			E_PML_Command.Suspend:
				stModeStateOut.RequestedState := E_PML_State.Suspended;
			
			E_PML_Command.Unsuspend:
				stModeStateOut.RequestedState := E_PML_State.Execute;
			
			E_PML_Command.Abort:
				stModeStateOut.RequestedState := E_PML_State.Aborted;
			
			E_PML_Command.Clear:
				stModeStateOut.RequestedState := E_PML_State.Stopped;
			
			E_PML_Command.Complete:
				stModeStateOut.RequestedState := E_PML_State.Complete;
			
		END_CASE

		// Wait done
		IF ((stModeStateOut.RequestedState = eCurrentState) AND (stModeStateOut.ModeStateResponse <= 0)) THEN
			// Set change status
			stModeStateOut.ChangeStatus := stModeStateIn.ChangeRequest;
			stModeStateOut.ModeStateResponse := 3;
			stModeStateOut.DataChange := stModeStateOut.DataChange + 1;
			stModeStateIn.State := E_PML_Command.Undefined;
			eCommand := E_PML_Command.Undefined;
		END_IF
	END_IF
END_IF


// Run State Machine
M_PackML_StateMachine();


// Update current mode/state
IF (DINT_TO_UINT(eCurrentMode) <> stModeStateOut.CurrentMode) THEN
	stModeStateOut.CurrentMode := DINT_TO_UINT(eCurrentMode);
	stModeStateOut.DataChange := stModeStateOut.DataChange + 1;	
END_IF
IF (DINT_TO_UINT(eCurrentState) <> stModeStateOut.CurrentState) THEN
	stModeStateOut.CurrentState := DINT_TO_UINT(eCurrentState);
	stModeStateOut.DataChange := stModeStateOut.DataChange + 1;	
END_IF

/// Static state "Aborted"
/// Trigged by "StateCompleted" when in "Aborting" state
/// Requires "Clear" to go to "Clearing" state 
{attribute 'object_name' := 'M_Aborted'}
METHOD M_Aborted
END_METHOD

/// Dynamic state "Aborting"
/// Trigged by "Abort" command
/// Requires "StateCompleted" to go to "Aborted" state 
{attribute 'object_name' := 'M_Aborting'}
METHOD M_Aborting
M_StateComplete();
END_METHOD

/// Set job data for mechanical roughing
METHOD PROTECTED M_CheckJobData : BOOL
VAR
	i						: UINT;
	bDynamicToolFound		: ARRAY [1..3] OF BOOL;		// Required Dynamic Tool(s) found
	bStationaryToolFound	: ARRAY [1..3] OF BOOL;		// Required Stationary Tool(s) found
	bDynamicMaterialFound	: ARRAY [1..3] OF BOOL;		// Required Dynamic Material(s) found
	bStationaryMaterialFound: ARRAY [1..3] OF BOOL;		// Required Stationary Material(s) found
END_VAR

// Check Job Type
// Should be overwritten in inherited FB's if JobData need to be checked!
M_CheckJobData := TRUE;
END_METHOD

/// Dynamic state "Clearing"
/// Trigged by "Clear" command "Aborted" state
/// Requires "StateCompleted" to go to "Stopped" state 
{attribute 'object_name' := 'M_Clearing'}
METHOD M_Clearing
M_StateComplete();
END_METHOD

/// Static state "Complete"
/// Trigged by "StateCompleted" when in "Completing" state
/// Requires "Reset" to go to "Resetting" state 
{attribute 'object_name' := 'M_Complete'}
METHOD M_Complete
END_METHOD

/// Dynamic state "Completing"
/// Trigged by "StageCompleted" command when in "Execute" state
/// Requires "StateCompleted" to go to "Complete" state 
{attribute 'object_name' := 'M_Completing'}
METHOD M_Completing
M_StateComplete();
END_METHOD

METHOD M_ErrorWarningObj : BOOL
VAR_INPUT
	bActive				: BOOL;
	iErrorWarningType	: UINT;
	diErrorWarningID 	: UDINT;
	sDeviceID			: STRING(30);
	iSeverity			: UINT;
	iNativeID			: UDINT;
	sNativeMessage		: STRING(80);
END_VAR
VAR_IN_OUT
	arErrorWaringData	: ARRAY [1..255] OF ST_ErrorWarningDataX;
END_VAR
VAR
	iFoundPos			: UINT;
	i					: UINT;
	j					: UINT;
END_VAR
//Look through array to find existing record(s)
FOR i := 1 TO 255 DO
	IF arErrorWaringData[i].ErrorWarningID = 0 THEN
		EXIT;
	END_IF
	//Existing alarm - first
	IF arErrorWaringData[i].ErrorWarningID = diErrorWarningID AND iFoundPos = 0 THEN
		iFoundPos := i;
	//Multiple records - delete
	ELSIF arErrorWaringData[i].ErrorWarningID = diErrorWarningID AND iFoundPos <> 0 THEN
		MEMSET(ADR(arErrorWaringData[i]), 0, SIZEOF(arErrorWaringData[i]));
		M_ErrorWarningObj := TRUE;
	END_IF
END_FOR

//Alarm high
IF bActive THEN
	//New alarm
	IF iFoundPos = 0 THEN
		arErrorWaringData[i].ErrorWarningType := iErrorWarningType;
		arErrorWaringData[i].DeviceID := sDeviceID;
		arErrorWaringData[i].Severity := iSeverity;
		arErrorWaringData[i].NativeID := iNativeID;
		arErrorWaringData[i].NativeMessage := sNativeMessage;
		arErrorWaringData[i].ErrorWarningID := diErrorWarningID;
		arErrorWaringData[i].DateTime := SYSTEMTIME_TO_STRING(fbGetTime.TIMESTR);
		M_ErrorWarningObj := TRUE;
	END_IF
	
//Alarm low
ELSIF NOT bActive AND iFoundPos <> 0 THEN
	MEMSET(ADR(arErrorWaringData[iFoundPos]), 0, SIZEOF(arErrorWaringData[iFoundPos]));
	M_ErrorWarningObj := TRUE;
END_IF

//Defrag
IF M_ErrorWarningObj THEN
	FOR i:= 1 TO 254 DO
		//Find first empty spot
		IF arErrorWaringData[i].ErrorWarningID = 0 THEN
			//Find first record
			FOR j:= i TO 255 DO
				IF arErrorWaringData[j].ErrorWarningID <> 0 THEN
					//Move to empty spot
					arErrorWaringData[i] := arErrorWaringData[j];
					MEMSET(ADR(arErrorWaringData[j]), 0, SIZEOF(arErrorWaringData[j]));
					EXIT;
				END_IF
			END_FOR
		END_IF
		//No more records
		IF j >= 255 THEN
			RETURN;
		END_IF
	END_FOR
END_IF
END_METHOD

/// Static state "Execute"
/// Trigged by "StageCompleted" when in "Starting" state
/// Trigged by "StageCompleted" when in "Unholding" state
/// Trigged by "StageCompleted" when in "Unsuspending" state
/// Requires "Hold" command to go to "Holding" state 
/// Requires "Suspend" command to go to "Suspending" state 
/// Requires "StageCompleted" to go to "Completing" state 
{attribute 'object_name' := 'M_Execute'}
METHOD M_Execute
M_StateComplete();
END_METHOD

/// Static state "Held"
/// Trigged by "StateCompleted" when in "Holding" state
/// Requires "Unhold" command to go to "Unholding" state 
{attribute 'object_name' := 'M_Held'}
METHOD M_Held
END_METHOD

/// Dynamic state "Holding"
/// Trigged by "Hold" command when in "Execute" state
/// Requires "StateCompleted" to go to "Held" state 
{attribute 'object_name' := 'M_Holding'}
METHOD M_Holding
M_StateComplete();
END_METHOD

/// Static state "Idle"
/// Trigged by "StateCompleted" when in "Resetting" state
/// Requires "Start" command to go to "Starting" state 
{attribute 'object_name' := 'M_Idle'}
METHOD M_Idle
END_METHOD

METHOD PROTECTED M_Init : BOOL
VAR_INPUT
END_VAR
IF (NOT bInitDone) THEN
	
	// OEE initial values
	stOEE.GoodProduct := iGoodProduct;	
	stOEE.RejectedProduct := iRejectedProduct;	
	stOEE.ProcessedProduct := iProcessedProduct;	

	bInitDone := TRUE;

END_IF
M_Init := bInitDone;
END_METHOD

METHOD PROTECTED M_OEEProductProcessed
VAR_INPUT
	bGood		: BOOL;
END_VAR

// Increment OEE values
iProcessedProduct := iProcessedProduct + 1;
stOEE.ProcessedProduct := iProcessedProduct;
IF (bGood) THEN
	iGoodProduct := iGoodProduct + 1;
	stOEE.GoodProduct := iGoodProduct;
ELSE
	iRejectedProduct := iRejectedProduct + 1;
	stOEE.RejectedProduct := iRejectedProduct;
END_IF

// TODO!!!
// Update Event ID!
stOEE.EventID;

// Update time for changes
stOEE.DateTime := SYSTEMTIME_TO_DT(TIMESTR := fbGetTime.TIMESTR);

// Increment DataChange to signal to LC that sometihng has changed
stOEE.DataChange := stOEE.DataChange + 1;
END_METHOD

METHOD PROTECTED M_PackML_StateMachine : BOOL
VAR_INPUT
END_VAR

CASE nStateModeChange OF

	0:	// Waiting for user request
		IF (NOT UnitModeChangeInProcess) THEN
			// Local unit mode change request
			IF (bProductionLocal AND (eCurrentMode <> Tc3_PackML_V2.ePMLProtUnitMode_Production)) THEN
				eMode := E_PML_Mode.Production;
				UnitModeChangeRequest := TRUE;
			ELSIF (bManualLocal AND (eCurrentMode <> Tc3_PackML_V2.ePMLProtUnitMode_Manual)) THEN
				eMode := E_PML_Mode.Manual;
				UnitModeChangeRequest := TRUE;
			ELSIF (bMaintenanceLocal AND (eCurrentMode <> Tc3_PackML_V2.ePMLProtUnitMode_Maintenance)) THEN
				eMode := E_PML_Mode.Maintenance;
				UnitModeChangeRequest := TRUE;
			END_IF
		END_IF
		bChangeIntoProduction := FALSE;
		IF ((eMode = ePMLProtUnitMode_Production) AND (eCurrentMode = ePMLProtUnitMode_Invalid)) THEN
			nStateModeChange := 1;
		ELSIF (UnitModeChangeRequest AND (eMode <> ePMLProtUnitMode_Production)) THEN
			nStateModeChange := 1;
		ELSIF ((eMode = ePMLProtUnitMode_Production) AND (eCurrentMode <> ePMLProtUnitMode_Production)) THEN
			nStateModeChange := 3;
		END_IF
		
	1:	// Starting UnitModeManager 
		fbUnitModeManager.bExecute := TRUE;
		fbUnitModeManager.eModeCommand := eMode;
		UnitModeChangeInProcess := TRUE;
	
		IF (fbUnitModeManager.bDone) THEN
			fbUnitModeManager.bExecute := FALSE;
			bInvalidModeCommandOut := FALSE;
			nStateModeChange := 0;
			bChangeIntoProduction := FALSE;
			UnitModeChangeInProcess := FALSE;
		ELSIF (fbUnitModeManager.bError) THEN
			bInvalidModeCommandOut := TRUE;
			fbUnitModeManager.bExecute := FALSE;
			nLastState := eCurrentState;
			nStateModeChange := 2;
			bChangeIntoProduction := FALSE;
			UnitModeChangeInProcess := FALSE;
		END_IF
	
	2:	// ErrorHanddling
		IF (bModeChangeRequest) THEN
			nStateModeChange := 0;
			bInvalidModeCommandOut := FALSE;
		ELSIF (nLastState <> eCurrentState) THEN
			bInvalidModeCommandOut := FALSE;
		END_IF
		
	3:	// state to check, if command 'Production' is valid
		IF ((eCurrentState = ePMLState_Aborted) OR (eCurrentState = ePMLState_Stopped) OR (eCurrentState = ePMLState_Idle)) THEN
			bChangeIntoProduction := TRUE;
			nStateModeChange := 1;
		ELSE
			nStateModeChange := 2;
			bInvalidModeCommandOut := TRUE;
			nLastState := eCurrentState;
		END_IF
END_CASE


// Run Unit Mode Manager
fbUnitModeManager(	eState := eCurrentState,
					eModeStatus => eCurrentMode,
					bDone => ,
					bError => ,
					nErrorId => 	);

IF (fbUnitModeManager.eModeStatus <> 0) THEN
	// Local E-stop/abort handling	
	IF (NOT bEStopOK OR bAbortLocal) THEN
		eCommand := DINT_TO_UINT(E_PMLCommand.ePMLCommand_Abort);
	END_IF
	// Local Start handling
	IF (bStartLocal) THEN
		eCommand := DINT_TO_UINT(E_PMLCommand.ePMLCommand_Start);
	END_IF
	// Local Stop handling
	IF (bStopLocal) THEN
		eCommand := DINT_TO_UINT(E_PMLCommand.ePMLCommand_Stop);
	END_IF
	// Local Reset handling
	IF (bResetLocal) THEN
		eCommand := DINT_TO_UINT(E_PMLCommand.ePMLCommand_Reset);
	END_IF
	// Local Clear handling
	IF (bClearLocal) THEN
		eCommand := DINT_TO_UINT(E_PMLCommand.ePMLCommand_Clear);
	END_IF
	// Local Hold handling
	IF (bHoldLocal) THEN
		eCommand := DINT_TO_UINT(E_PMLCommand.ePMLCommand_Hold);
	END_IF
	// Local Unhold handling
	IF (bUnholdLocal) THEN
		eCommand := DINT_TO_UINT(E_PMLCommand.ePMLCommand_Unhold);
	END_IF
	// Local Suspend handling
	IF (bSuspendLocal) THEN
		eCommand := E_PMLCommand.ePMLCommand_Suspend;
	END_IF
	// Local Unsuspend handling
	IF (bSuspendLocal) THEN
		eCommand := E_PMLCommand.ePMLCommand_Unsuspend;
	END_IF
	
	// Calling the StateMachine, when there is a valid Mode
	fbStateMachine(	eMode := eCurrentMode,
					eCommand := eCommand,
					stSubUnitInfoRef := ,
					stOptions := ,
					eState => eCurrentState,
					bError => ,
					nErrorID => 	);

END_IF

// Requested state:
CASE eCommand OF			
	E_PMLCommand.ePMLCommand_Abort:
		eRequestedState := E_PMLState.ePMLState_Aborted;
		
	E_PMLCommand.ePMLCommand_Clear:
		eRequestedState := E_PMLState.ePMLState_Stopped;

	E_PMLCommand.ePMLCommand_Complete:
		eRequestedState := E_PMLState.ePMLState_Complete;
		
	E_PMLCommand.ePMLCommand_Hold:
		eRequestedState := E_PMLState.ePMLState_Held;
		
	E_PMLCommand.ePMLCommand_Reset:
		eRequestedState := E_PMLState.ePMLState_Idle;
		
	E_PMLCommand.ePMLCommand_Start:
		eRequestedState := E_PMLState.ePMLState_Execute;
		
	E_PMLCommand.ePMLCommand_Stop:
		eRequestedState := E_PMLState.ePMLState_Stopped;
		
	E_PMLCommand.ePMLCommand_Suspend:
		eRequestedState := E_PMLState.ePMLState_Suspended;
		
	E_PMLCommand.ePMLCommand_Unhold:
		eRequestedState := E_PMLState.ePMLState_Execute;
		
	E_PMLCommand.ePMLCommand_Unsuspend:
		eRequestedState := E_PMLState.ePMLState_Execute;
		
END_CASE


//One of the methods is executing by the actual state
CASE eCurrentState OF
	E_PML_State.Undefined:
		M_Undefined();
	E_PML_State.Clearing:
		M_Clearing();
	E_PML_State.Stopped:
		M_Stopped();
	E_PML_State.Starting:
		M_Starting();
	E_PML_State.Idle:
		M_Idle();
	E_PML_State.Suspended:
		M_Suspended();
	E_PML_State.Execute:
		M_Execute();
	E_PML_State.Stopping:
		M_Stopping();
	E_PML_State.Aborting:
		M_Aborting();
	E_PML_State.Aborted:
		M_Aborted();
	E_PML_State.Holding:
		M_Holding();
	E_PML_State.Held:
		M_Held();
	E_PML_State.Unholding:
		M_Unholding();
	E_PML_State.Suspending:
		M_Suspending();
	E_PML_State.Unsuspending:
		M_Unsuspending();
	E_PML_State.Resetting:
		M_Resetting();
	E_PML_State.Completing:
		M_Completing();
	E_PML_State.Complete:
		M_Complete();
END_CASE
END_METHOD

/// Dynamic state "Resetting"
/// Trigged by "Reset" command when in "Stopped" state
/// Requires "StateCompleted" to go to "Idle" state 
{attribute 'object_name' := 'M_Resetting'}
METHOD M_Resetting
M_StateComplete();
END_METHOD

/// Dynamic state "Starting"
/// Trigged by "Start" command when in "Idle" state
/// Requires "StateCompleted" to go to "Execute" state 
{attribute 'object_name' := 'M_Starting'}
METHOD M_Starting
M_StateComplete();
END_METHOD

{attribute 'object_name' := 'M_StateComplete'}
METHOD M_StateComplete
//the actual state is completed
fbStateMachine.M_StateComplete();
END_METHOD

/// Static state "Stopped"
/// Trigged by "StateCompleted" when in "Stopping" state
/// Requires "Reset" command to go to "Resetting" state 
{attribute 'object_name' := 'M_Stopped'}
METHOD M_Stopped
END_METHOD

/// Dynamic state "Stopping"
/// Trigged by "Stop" command
/// Requires "StateCompleted" to go to "Stopped" state 
{attribute 'object_name' := 'M_Stopping'}
METHOD M_Stopping
M_StateComplete();
END_METHOD

/// Static state "Suspended"
/// Trigged by "StateCompleted" when in "Suspending" state
/// Requires "Unsuspend" command to go to "Unsuspending" state 
{attribute 'object_name' := 'M_Suspended'}
METHOD M_Suspended
END_METHOD

/// Dynamic state "Suspending"
/// Trigged by "Suspend" command when in "Execute" state
/// Requires "StateCompleted" to go to "Suspended" state 
{attribute 'object_name' := 'M_Suspending'}
METHOD M_Suspending
M_StateComplete();
END_METHOD

{attribute 'object_name' := 'M_Undefined'}
METHOD M_Undefined
END_METHOD

/// Dynamic state "Unholding"
/// Trigged by "Unhold" command when in "Held" state
/// Requires "StateCompleted" to go to "Execute" state 
{attribute 'object_name' := 'M_Unholding'}
METHOD M_Unholding
M_StateComplete();
END_METHOD

/// Dynamic state "Unsuspending"
/// Trigged by "Unsuspend" command when in "Suspended" state
/// Requires "StateCompleted" to go to "Execute" state 
{attribute 'object_name' := 'M_Unsuspending'}
METHOD M_Unsuspending
M_StateComplete();
END_METHOD

END_FUNCTION_BLOCK

// ---- ECC/Tools/F_LogLine.TcPOU
FUNCTION F_LogLine : DINT
VAR_INPUT
	sLogString	: STRING(250);
	iValue		: DINT;
END_VAR
VAR
	iReplacePos	: INT;
	sLogFile	: STRING;
END_VAR

	// Log to output window as info message
	IF (bLogToOutputWindow) THEN
		F_LogLine:= ADSLOGDINT(ADSLOG_MSGTYPE_HINT OR ADSLOG_MSGTYPE_LOG,sLogString, iValue);
	END_IF
	
	// Replace the '%d' in the log string with the stinr-value of the iValue input 
	iReplacePos := FIND(sLogString, '%d');
	IF (iReplacePos > 0) THEN
		// '%d' found in string
		sLogFile := REPLACE(sLogString, DINT_TO_STRING(iValue), 2, iReplacePos);
	ELSE
		sLogFile := sLogString;
	END_IF

	// Log to file
	F_LogFile(sLogFile);

END_FUNCTION

// ---- ECC/Tools/LogToFile/F_LogFile.TcPOU
FUNCTION F_LogFile : BOOL
VAR_INPUT
	msg		: STRING(200);

END_VAR
VAR
	Temp:ULINT;
	CurrentDate:STRING(10);
	msgWithTime :STRING(200);
	DateTimeNow :STRING;
END_VAR

(* Get date and time *)

DateTimeNow  := SYSTEMTIME_TO_STRING(fbLocalTime.systemTime);

(* Set date to check for generation of new file *)
CurrentDate := DateTimeNow;

(* Add date and time to line of log *)
msgWithTime := CONCAT(DateTimeNow, ' ');
msgWithTime := CONCAT(msgWithTime, msg);
msgWithTime := CONCAT(msgWithTime, '$N');


(* Write to FIFO *)
IF LogToTextBuffer.Count <= LogToTextBuffer.DataTop THEN

	(* Calculate new insert pointer *)
	LogToTextBuffer.Input_Pointer := LogToTextBuffer.Input_Pointer + 1;
	IF LogToTextBuffer.Input_Pointer > LogToTextBuffer.DataTop THEN
		LogToTextBuffer.Input_Pointer := 0;
	END_IF

	(* If data is empty, sync output pointer *)
	IF LogToTextBuffer.Count = 0 THEN
		LogToTextBuffer.Output_Pointer := LogToTextBuffer.Input_Pointer;
	END_IF

	(* Store data *)
	LogToTextBuffer.DB[LogToTextBuffer.Input_Pointer] := msgWithTime;

	LogToTextBuffer.Count := LogToTextBuffer.Count + 1;
END_IF

END_FUNCTION

// ---- ECC/Cell_Unit_4/HeatAndSteamDeviceDriver/FB_EMS_HS.TcPOU
FUNCTION_BLOCK FB_EMS_HS
VAR_INPUT
END_VAR
VAR_OUTPUT
END_VAR
VAR
// ModBus data structures
	uRead			: U_EMS_HS_Read;
	uWrite			: U_EMS_HS_Write;
	
	// Modbus reading
	tonMBRead		: TON;		// Timer to handle reading requests from device
	fbMBRead		: Tc2_ModbusSrv.FB_MBReadRegs;	// FB for reading modbus register(s)
	bMBRead_Busy	: BOOL;
	bMBRead_Error	: BOOL;
	nMBRead_ErrorID	: UDINT;
	cbMBRead_Read	: UDINT;
	trigMBReadError	: R_TRIG;
	fbGetReadTime	: NT_GetTime;
	trigReadDone	: F_TRIG;
	tsLastRead		: TIMESTRUCT;
	iReads			: UINT;
	iErrorReads		: UINT;

// Modbus writing
	tonMBWrite		: TON;		// Timer to handle writing requests to device
	fbMBWrite		: Tc2_ModbusSrv.FB_MBWriteRegs;	// FB for writing modbus register(s)
	bMBWrite_Busy	: BOOL;
	bMBWrite_Error	: BOOL;
	nMBWrite_ErrorID: UDINT;
	trigWriteDone	: F_TRIG;
	trigMBWriteError: R_TRIG;
	fbGetWriteTime	: NT_GetTime;
	tsLastWrite		: TIMESTRUCT;
	iWrites			: UINT;
	iErrorWrites	: UINT;
	
//Local vars
	bAbortLocal 	: BOOL;
	bManualLocal	: BOOL;
	bProductionLocal: BOOL;
// Simulation
	bSimMode		: BOOL;	// TRUE if simulation should be used (no start device, no setpoints to device)
END_VAR
VAR PERSISTENT
	sIPAddr			: STRING(15);	// Station IP address
	tTimeout		: TIME := T#5S;
END_VAR


// Simulation mode ?
// Only perform communication if NOT in simulation mode
IF (NOT M_Simulation()) THEN

	// Device controller
	M_ModBusRead(	rInterval := 1,
					wAddress := 2501,
					wNoOfRegisters := 23,
					pbDestAddress := ADR(uRead.aWords),
					dwDestSize := SIZEOF(uRead.aWords)	);
	
	M_ModBusWrite(	rInterval := 1, 
					wAddress := 2601,
					wNoOfRegisters := 8,	
					pbSrcAddress := ADR(uWrite.aWords),
					dwSrcSize := SIZEOF(uWrite.aWords)	);
END_IF

// Local state changes
IF (uRead.stVars.eMachStatus = E_EMS_HS_Status.ALARM) THEN
	bAbortLocal := TRUE;
ELSIF (uRead.stVars.stStates.ALARM_IN_PROGRESS) THEN
	bAbortLocal := TRUE;
ELSIF (NOT uRead.stVars.stStates.REMOTE_MODE) THEN
	bAbortLocal := TRUE;
ELSE
	bAbortLocal := FALSE;
END_IF
IF (NOT uRead.stVars.stStates.REMOTE_MODE) THEN
	bManualLocal := TRUE;
	bProductionLocal := FALSE;
ELSE
	bProductionLocal := TRUE;
	bManualLocal := FALSE;
END_IF

METHOD PROTECTED M_CmdNeutral : BOOL
VAR_INPUT
END_VAR
uWrite.stVars.stCommands.REMOTE_START := FALSE;
uWrite.stVars.stCommands.REMOTE_STOP := FALSE;
END_METHOD

METHOD PROTECTED M_Cmdreset : BOOL
VAR_INPUT
END_VAR
END_METHOD

METHOD PROTECTED M_CmdStart : BOOL
VAR_INPUT
END_VAR
uWrite.stVars.stCommands.REMOTE_START := TRUE;
uWrite.stVars.stCommands.REMOTE_STOP := FALSE;
END_METHOD

METHOD PROTECTED M_CmdStop : BOOL
VAR_INPUT
END_VAR
uWrite.stVars.stCommands.REMOTE_START := FALSE;
uWrite.stVars.stCommands.REMOTE_STOP := TRUE;
END_METHOD

/// Read modbus TCP register(s)
METHOD PROTECTED M_ModBusRead : BOOL
VAR_INPUT
	rInterval		: REAL;
	wAddress		: WORD;				// Register address to read
	wNoOfRegisters	: WORD;				// Register to read from station
	pbDestAddress	: POINTER TO BYTE;	// Address of mem to place read data
	dwDestSize		: DWORD;			// Size of mem to place read data
END_VAR
// Timer
tonMBRead(	IN := NOT tonMBRead.Q,
			PT := REAL_TO_TIME(rInterval * 1000.0),
			Q => 	);

// Read data from device via. modbus TCP
fbMBRead(	sIPAddr:= sIPAddr, 				// Station IP address
			nTCPPort:= MODBUS_TCP_PORT, 	// Modbus TCP port (normally 502)
			nUnitID:= 1,//16#FF, 			// If a device is addressed directly via TCP/IP, this value must be 16#FF.
			nQuantity:= wNoOfRegisters,		// Number of words (registers) to read 
			nMBAddr:= wAddress - 1,			// Addres of registers to read ( -1 needed ) 
			cbLength:= dwDestSize,			// Contains the max. byte size of the destination buffer. The minimum buffer byte size must be: nQuantity * 2.
			pDestAddr:= pbDestAddress, 		// Address of the destination buffer into which the data are to be read.
			bExecute:= tonMBRead.Q,			// Trig reading
			tTimeout:= tTimeout, 			// States the length of the timeout that may not be exceeded by execution of the ADS command
			bBusy=> bMBRead_Busy, 
			bError=> bMBRead_Error, 
			nErrId=> , 
			cbRead=> cbMBRead_Read);

// Last read time
trigReadDone(CLK := (fbMBRead.bBusy AND NOT fbMBRead.bError));
trigMBReadError(CLK := bMBRead_Error);
IF (trigReadDone.Q) THEN
	iReads := iReads + 1;
END_IF
IF (trigMBReadError.Q) THEN
	iErrorReads := iErrorReads + 1;
	nMBRead_ErrorID := fbMBRead.nErrId;
END_IF
fbGetReadTime(	NETID:= '', 
				START:= trigReadDone.Q,
				TMOUT:= T#5S, 
				BUSY=> , 
				ERR=> , 
				ERRID=> , 
				TIMESTR=> tsLastRead);

// Station communication status
M_ModBusRead := (cbMBRead_Read = wNoOfRegisters * 2);
END_METHOD

/// Writes ModBus TCP registers
METHOD PROTECTED M_ModBusWrite : BOOL
VAR_INPUT
	rInterval		: REAL;
	wAddress		: WORD;				// Register address to write to
	wNoOfRegisters	: WORD;				// Register(s) to write to station
	pbSrcAddress	: POINTER TO BYTE;	// Address of mem to read source data from
	dwSrcSize		: DWORD;			// Size of mem to read source data from
END_VAR
VAR
END_VAR
// Timer
tonMBWrite(	IN := NOT tonMBWrite.Q,
			PT := REAL_TO_TIME(rInterval * 1000.0),
			Q => 	);

// Write data to device via. modbus TCP
fbMBWrite(	sIPAddr:= sIPAddr, 				// Station IP address
			nTCPPort:= MODBUS_TCP_PORT, 	// Modbus TCP port (normally 502)
			nUnitID:= 1,//16#FF, 			// If a device is addressed directly via TCP/IP, this value must be 16#FF.
			nQuantity:= wNoOfRegisters,		// Number of words (registers) to write 
			nMBAddr:= wAddress - 1,			// Addres of registers to write 
			cbLength:= dwSrcSize,			// Contains the max. byte size of the source buffer. The minimum buffer byte size must be: nQuantity * 2.
			pSrcAddr:= pbSrcAddress,	 	// Address of the source buffer from which, the data are read
			bExecute:= tonMBWrite.Q,		// Trig writing 
			tTimeout:= tTimeout, 			// States the length of the timeout that may not be exceeded by execution of the ADS command
			bBusy=> bMBWrite_Busy, 
			bError=> bMBWrite_Error, 
			nErrId=> );

// Last write time
trigWriteDone(CLK := (fbMBWrite.bBusy AND NOT fbMBWrite.bError));
trigMBWriteError(CLK := bMBWrite_Error);
IF (trigWriteDone.Q) THEN
	iWrites := iWrites + 1;
END_IF
IF (trigMBWriteError.Q) THEN
	iErrorWrites := iErrorWrites + 1;
	nMBWrite_ErrorID := fbMBWrite.nErrId;
END_IF
fbGetWriteTime(	NETID:= '', 
				START:= trigWriteDone.Q,
				TMOUT:= T#5S, 
				BUSY=> , 
				ERR=> , 
				ERRID=> , 
				TIMESTR=> tsLastWrite);

// Station communication status
M_ModBusWrite := trigWriteDone.Q;
END_METHOD

METHOD PROTECTED M_Simulation : BOOL
VAR_INPUT
END_VAR

IF (bSimMode) THEN
	// Simulation mode ENABLED

	// Device start command
	IF (uWrite.stVars.stCommands.REMOTE_START) THEN
		// Device states
		uRead.stVars.eMachStatus := E_EMS_HS_Status.READY;
		uRead.stVars.stStates.MACHINE_READY_TO_WORK := TRUE;
		uRead.stVars.stStates.TEMP_START_BELT_REACHED := TRUE;
		uRead.stVars.stStates.TEMP_START_STEAM_REACHED := TRUE;
		uRead.stVars.stStates.MACHINE_IN_STANDBY := FALSE;
		// Device temperature
		uRead.stVars.rActTempVal := uWrite.stVars.rSetTemp;
	ELSE
		// Device states
		uRead.stVars.eMachStatus := E_EMS_HS_Status.STANDBY;
		uRead.stVars.stStates.MACHINE_READY_TO_WORK := FALSE;
		uRead.stVars.stStates.TEMP_START_BELT_REACHED := FALSE;
		uRead.stVars.stStates.TEMP_START_STEAM_REACHED := FALSE;
		uRead.stVars.stStates.MACHINE_IN_STANDBY := TRUE;
	END_IF
	// Temperature setpoint value
	uRead.stVars.rActTempSetpoint := uWrite.stVars.rSetTemp;
	// Steam setpoint value
	uRead.stVars.rActSteamReq := uWrite.stVars.rSetSteamReq;
	// Fan setpoint value
	uRead.stVars.rActFanReq := uWrite.stVars.rSetFanSpeed;
	// Alarms
	uRead.stVars.stAlarms.TEMP_PROBE_FAULT := FALSE;
	uRead.stVars.stAlarms.FAULT_INVERTER := FALSE;
	uRead.stVars.stAlarms.ENERGY_METER_COM_ERROR := FALSE;
	// Device states
	uRead.stVars.stStates.REMOTE_MODE := TRUE;
	uRead.stVars.stStates.ALARM_IN_PROGRESS := FALSE;
	uRead.stVars.stStates.MACHINE_IN_HEATING := FALSE;
	
	M_Simulation := TRUE;

ELSE
	// Simulation mode DISABLED

	M_Simulation := FALSE;

END_IF
END_METHOD

METHOD PROTECTED M_StaAlarm : BOOL
VAR_INPUT
END_VAR
M_StaAlarm := (uRead.stVars.eMachStatus = E_EMS_HS_Status.ALARM);
END_METHOD

METHOD PROTECTED M_StaReady : BOOL
VAR_INPUT
END_VAR
M_StaReady := (uRead.stVars.eMachStatus = E_EMS_HS_Status.READY);
END_METHOD

METHOD PROTECTED M_StaStandby : BOOL
VAR_INPUT
END_VAR
M_StaStandby := (uRead.stVars.eMachStatus = E_EMS_HS_Status.STANDBY);
END_METHOD

PROPERTY PUBLIC P_bSimulationMode : BOOL
GET
P_bSimulationMode := bSimMode;
END_GET
SET
bSimMode := P_bSimulationMode;
END_SET
END_PROPERTY

PROPERTY P_ModbusIPBarrera : STRING
GET
P_ModbusIPBarrera := sIPAddr;
END_GET
SET
sIPAddr := P_ModbusIPBarrera;
END_SET
END_PROPERTY

PROPERTY PUBLIC P_rSetFanSpeed : REAL
SET
uWrite.stVars.rSetFanSpeed := P_rSetFanSpeed;
END_SET
END_PROPERTY

PROPERTY PUBLIC P_rSetSteamReq : REAL
SET
uWrite.stVars.rSetSteamReq := REAL_TO_DINT(P_rSetSteamReq);
END_SET
END_PROPERTY

PROPERTY PUBLIC P_rSetTemp : REAL
SET
uWrite.stVars.rSetTemp := P_rSetTemp;
END_SET
END_PROPERTY

PROPERTY PUBLIC P_stCellCommandData : ST_EMS_HS_Write
GET // PUBLIC
P_stCellCommandData := uWrite.stVars;
END_GET
SET // PUBLIC
uWrite.stVars := P_stCellCommandData;
END_SET
END_PROPERTY

PROPERTY PUBLIC P_stCellStatusData : ST_EMS_HS_Read
GET
P_stCellStatusData := uRead.stVars;
END_GET
END_PROPERTY

END_FUNCTION_BLOCK

// ---- ECC/Tools/F_StringCompNoCase.TcPOU
FUNCTION F_StringCompNoCase : BOOL
VAR_INPUT
	s1		: STRING;
	s2		: STRING;
END_VAR
VAR
END_VAR


F_StringCompNoCase := ( F_ToUCase(s1) = F_ToUCase(s2) );

END_FUNCTION

// ---- ECC/Basic/OPC Data/F_NewDeviceDataX.TcPOU
FUNCTION F_NewDeviceDataX : ST_DeviceDataX
VAR_INPUT
	sDeviceID			: STRING;			// The ID of the specific device
	sDeviceName			: STRING;			// The descriptive name of the device
	iDataID				: UDINT;			// The ID of the operational data
	sDataName			: STRING;			// The descriptive name of the operational data
	eUnit				: E_Units;	// The symbolic description of the measuring unit
END_VAR
VAR
END_VAR

// Create structure

F_NewDeviceDataX.DeviceID := sDeviceID;
F_NewDeviceDataX.DeviceName :=sDeviceName;
F_NewDeviceDataX.DataID := iDataID;
F_NewDeviceDataX.DataName := sDataName;
F_NewDeviceDataX.UnitID := Units.Code(eUnit);	// Extracts common unit code from pre-defined unit types
F_NewDeviceDataX.Unit := Units.Text(eUnit);		// Extracts common unit symbol from pre-definded unit types

END_FUNCTION

// ---- ECC/Cell_Unit_4/HeatAndSteam/F_CalcValuesHeatSteam.TcPOU
FUNCTION F_CalcValuesHeatSteam : REAL
VAR_INPUT
	rTempFinal		: REAL;				// [°C]		
	rTempInitial	: REAL;				// [°C]		
	rCT				: REAL;				// []		Coefficient for temperature
	rCS				: REAL;				// []		Coefficient for steam
	rCA				: REAL;				// []		Coefficient for airflow
	rMachineLength	: REAL;				// [m]		Length of machine
	// Limits
	rTimeMin		: REAL;				// [s]		Minimum allowed time in machine
	rTimeMax		: REAL;				// [s]		Maximum allowed time in machine
	rTempMin		: REAL;				// [°C]		Minimum allowed temperature in machine
	rTempMax		: REAL;				// [°C]		Maximum allowed temperature in machine
	rSteamMin		: REAL;				// []		Minimum allowed steam in machine
	rSteamMax		: REAL;				// []		Maximum allowed steam in machine
	rAirMin			: REAL;				// []		Minimum allowed airflow in machine
	rAirMax			: REAL;				// []		Maximum allowed airflow in machine	
END_VAR
VAR_OUTPUT
	rVelocity		: REAL;				// [m/s]	Carrier velocity
	rTempMachine	: REAL;				// [°C]		Machine temperature
	rTimeMachine	: REAL;				// [s]		Time in machine
	rSteamMachine	: REAL;				// []		
	rAirMachine		: REAL;				// []		
END_VAR
VAR
	// Limits
	rVelocityMin	: REAL := 0.001;	// [m/s]	Minimum allowed speed
	rVelocityMax	: REAL := 2.0;		// [m/s]	Maximum allowed speed
	
	// Temp
	rVelocityCalcRaw: REAL;				// [m/s]	
	rVelocityCalc	: REAL;				// [m/s]	
	rTimeCalcRaw	: REAL;				// [s]		
	rTimeCalc		: REAL;				// [s]		
	sTempString		: STRING(200);		// 			
END_VAR


// Calculate time needed in device and machine temperature
//t = ( (TFinal) / (TMachine * cT + SMachine * cS + AMachine * cA) ) - TInitial

// If constants are ZERO use fixed time in mechine from job data (minimum time)
IF ( (rCT = 0.0) AND (rCS = 0.0) AND (rCA = 0.0) ) THEN
	rTimeCalcRaw := rTimeMin;
	rTempMachine := rTempMax;
	rSteamMachine := rSteamMax;
	rAirMax := rAirMax;
	
ELSE
	rTempMachine := (rTempMin + rTempMax) / 2.0;
	rSteamMachine := (rSteamMin + rSteamMax) / 2.0;
	rAirMachine := (rAirMin + rAirMax) / 2.0;

	// Check for divide-by-zero
	IF ((rTempMachine * rCT) + (rSteamMachine * rCS) + (rAirMachine * rCA)) = 0.0 THEN
		rTimeCalcRaw := rTimeMin;
		rTempMachine := rTempMax;
		rSteamMachine := rSteamMax;
		rAirMax := rAirMax;
	ELSE
		rTimeCalcRaw := (rTempFinal - rTempInitial) / ((rTempMachine * rCT) + (rSteamMachine * rCS) + (rAirMachine * rCA));	
	END_IF
	
END_IF

// Limit time in device according to job data
rTimeCalc := LIMIT(rTimeMin, rTimeCalcRaw, rTimeMax);

// Make sure time is not ZERO
IF (rTimeCalc <= 0.0) THEN
	rTimeCalc := 120.0;

END_IF

// Calculate velocity based on time in machine and machine length
rVelocityCalcRaw := rMachineLength / rTimeCalc;

// Limit velocity to allowed limits
rVelocityCalc := LIMIT(rVelocityMin, rVelocityCalcRaw, rVelocityMax);

// Log
	sTempString := CONCAT('STAT: ', 'Velocity Calc ');
	sTempString := CONCAT(sTempString, '. Temp=');
	sTempString := CONCAT(sTempString, TO_STRING(rTempMachine));
	sTempString := CONCAT(sTempString, '. Steam=');
	sTempString := CONCAT(sTempString, TO_STRING(rSteamMachine));
	sTempString := CONCAT(sTempString, '. Air=');
	sTempString := CONCAT(sTempString, TO_STRING(rAirMachine));
	sTempString := CONCAT(sTempString, '. Time_RAW=');
	sTempString := CONCAT(sTempString, TO_STRING(rTimeCalcRaw));
	sTempString := CONCAT(sTempString, '. Time=');
	sTempString := CONCAT(sTempString, TO_STRING(rTimeCalc));
	sTempString := CONCAT(sTempString, '. Vel_RAW=');
	sTempString := CONCAT(sTempString, TO_STRING(rVelocityCalcRaw));
	sTempString := CONCAT(sTempString, '. Vel=');
	sTempString := CONCAT(sTempString, TO_STRING(rVelocityCalc));
	F_Logfile(sTempString);

// Output
rVelocity := rVelocityCalc;
rTempMachine := rTempMachine;
rSteamMachine := rSteamMachine;
rAirMachine := rAirMachine;
rTimeMachine := rTimeCalc;

END_FUNCTION

// ---- ECC/Cell_Unit_4/HeatAndSteam/FB_HeatAndSteamOUT.TcPOU
FUNCTION_BLOCK FB_HeatAndSteamOUT EXTENDS FB_Station_Basic
VAR_INPUT
END_VAR
VAR_OUTPUT
END_VAR
VAR_IN_OUT
	// Inputs
	stJobDataIn				: ST_InputStationHSJobData;
	stConfigIn				: ST_InputStationHSConfiguration;
	stUpcomingConfigIn		: ST_InputStationHSUpcomingConfiguration;
	stControlIn				: ST_InputStationHSControl;
	stAdditionalDataIn		: ST_InputStationHSAdditionalData;
	// Outputs
	stJobDataOut			: ST_OutputStationHSJobData;
	stConfigOut				: ST_OutputStationHSCurrentConfiguration;
	stUpcomingConfigOut		: ST_OutputStationHSUpcomingConfiguration;
	stOperationalDataOut	: ST_OutputStationHSOperationalData;
	stSustainabilityData	: ST_OutputStationHSSustainabilityData;
	stAdditionalDataOut		: ST_OutputStationHSAdditionalData;	
END_VAR 
VAR
	iOldChangeRequest		: UINT;

// Start up
	nCheckValid				: UINT;

END_VAR

SUPER^( stModeStateIn := stModeStateIn,
		stModeStateOut := stModeStateOut,
		stOEE := stOEE,
		stErrorWarning := stErrorWarning);

M_Init();

//Automatic reset when operation complete
bResetLocal := (eCommand <> ePMLCommand_Start AND eCurrentState = E_PMLState.ePMLState_Complete);

/// Static state "Aborted"
/// Trigged by "StateCompleted" when in "Aborting" state
/// Requires "Clear" to go to "Clearing" state 
{attribute 'object_name' := 'M_Aborted'}
METHOD M_Aborted
END_METHOD

/// Dynamic state "Aborting"
/// Trigged by "Abort" command
/// Requires "StateCompleted" to go to "Aborted" state 
{attribute 'object_name' := 'M_Aborting'}
METHOD M_Aborting
// Stop all moving parts
(* STOP all OPSTIONS and Track - Clear alarms og gå til Complete*)

M_StateComplete();
END_METHOD

METHOD M_ClearAll : BOOL
VAR_INPUT
END_VAR

IF eCurrentState = E_PMLState.ePMLState_Aborted OR eCurrentState = E_PMLState.ePMLState_Aborting THEN
	
	F_Logfile('ST2 - All data cleared!');
	
	M_ClearAll := TRUE;
END_IF
END_METHOD

/// Dynamic state "Clearing"
/// Trigged by "Clear" command "Aborted" state
/// Requires "StateCompleted" to go to "Stopped" state 
{attribute 'object_name' := 'M_Clearing'}
METHOD M_Clearing
(* Clear all OPSTIONS and Track - Clear alarms og gå til Complete*)

M_StateComplete();
END_METHOD

/// Static state "Complete"
/// Trigged by "StateCompleted" when in "Completing" state
/// Requires "Reset" to go to "Resetting" state 
{attribute 'object_name' := 'M_Complete'}
METHOD M_Complete
END_METHOD

/// Dynamic state "Completing"
/// Trigged by "StageCompleted" command when in "Execute" state
/// Requires "StateCompleted" to go to "Complete" state 
{attribute 'object_name' := 'M_Completing'}
METHOD M_Completing

VAR
	
END_VAR

// Reset execute sequence
// Job status data to OPC 

//Store old data for comparison



M_StateComplete();
END_METHOD

METHOD M_ConfigurationHandling
VAR_INPUT
END_VAR
VAR
	sTempSTring		: STRING(200);
END_VAR
// Is updated from operator/HMI
IF (stConfigIn.ChangeRequest <> stConfigOut.ChangeStatus) AND (stConfigIn.ChangeRequest > 0) THEN
	sTempString := CONCAT('Station 2 - ConfigChange request - Old request: ', TO_STRING(stConfigOut.ChangeStatus));
	sTempString := CONCAT(sTempString, ', New request: ');
	sTempString := CONCAT(sTempString, TO_STRING(stConfigIn.ChangeRequest));
	sTempString := CONCAT(sTempString, ' ConfigType: ');
	F_LogFile(CONCAT(sTempString, stConfigIn.ConfigurationType)); 
	
	// Change request from Line Controller
	stConfigOut.ChangeAcknowledge := stConfigIn.ChangeRequest;
	
	// Check Configuration Type
	IF (stConfigIn.ConfigurationType = 'OP11600') THEN	
		// Update output job data
		stConfigOut.ConfigurationType := stConfigIn.ConfigurationType;
		stConfigOut.DateTime := SYSTEMTIME_TO_DT(timestr:=fbGetTime.TIMESTR);
		stConfigOut.OP11600 := stConfigIn.OP11600;
		
		// Signal that job data has been written		
		stConfigOut.ChangeStatus := stConfigIn.ChangeRequest;
		
		// Signal that output job data has been updated
		stConfigOut.DataChange := stConfigOut.DataChange + 1;

	ELSE
		// Wrong configuration data type!
		stConfigOut.ConfigurationType := '';
		stConfigOut.DateTime := SYSTEMTIME_TO_DT(timestr:=fbGetTime.TIMESTR);

		// Signal that configuration data has been written		
		stConfigOut.ChangeStatus := stConfigIn.ChangeRequest;
		
		// Signal that output configuration data has been updated
		stConfigOut.DataChange := stConfigOut.DataChange + 1;

	END_IF
END_IF


// Upcoming Configuration
IF (stUpcomingConfigIn.ChangeRequest <> stUpcomingConfigOut.ChangeStatus) AND (stUpcomingConfigIn.ChangeRequest > 0) THEN
	sTempString := CONCAT('Station 2 Upcoming ConfigChange request - Old request: ', TO_STRING(stUpcomingConfigOut.ChangeStatus));
	sTempString := CONCAT(sTempString, ', New request: ');
	sTempString := CONCAT(sTempString, TO_STRING(stUpcomingConfigIn.ChangeRequest));
	sTempString := CONCAT(sTempString, ' ConfigType: ');
	F_LogFile(CONCAT(sTempString, stUpcomingConfigIn.ConfigurationType)); 	

	// Change request from Line Controller
	stUpcomingConfigOut.ChangeAcknowledge := stUpcomingConfigIn.ChangeRequest;
	
	// Check Configuration Type
	IF (stUpcomingConfigIn.ConfigurationType = 'OP11600') THEN	
		// Update configuration data
		stUpcomingConfigOut.ConfigurationType := stUpcomingConfigIn.ConfigurationType;
		stConfigOut.DateTime := SYSTEMTIME_TO_DT(timestr:=fbGetTime.TIMESTR);
		stUpcomingConfigOut.OP11600 := stUpcomingConfigIn.OP11600;

		// Signal that configuration data has been written		
		stUpcomingConfigOut.ChangeStatus := stUpcomingConfigIn.ChangeRequest;
		
		// Signal that output configuration data has been updated
		stUpcomingConfigOut.DataChange := stUpcomingConfigOut.DataChange + 1;
		
	ELSE
		// Wrong configuration data type!
		stUpcomingConfigOut.ConfigurationType := '';
		stConfigOut.DateTime := SYSTEMTIME_TO_DT(timestr:=fbGetTime.TIMESTR);

		// Signal that configuration data has been written		
		stUpcomingConfigOut.ChangeStatus := stUpcomingConfigIn.ChangeRequest;
		
		// Signal that output configuration data has been updated
		stUpcomingConfigOut.DataChange := stUpcomingConfigOut.DataChange + 1;

	END_IF
END_IF
END_METHOD

METHOD PROTECTED M_ErrorWarning
VAR_INPUT
END_VAR
VAR
END_VAR



// Alarms // TODO
END_METHOD

/// Static state "Execute"
/// Trigged by "StageCompleted" when in "Starting" state
/// Trigged by "StageCompleted" when in "Unholding" state
/// Trigged by "StageCompleted" when in "Unsuspending" state
/// Requires "Hold" command to go to "Holding" state 
/// Requires "Suspend" command to go to "Suspending" state 
/// Requires "StageCompleted" to go to "Completing" state 
{attribute 'object_name' := 'M_Execute'}
METHOD M_Execute

 M_StateComplete();
END_METHOD

METHOD M_ExternalStart
VAR_INPUT
END_VAR
bStartLocal := TRUE;
END_METHOD

/// Static state "Held"
/// Trigged by "StateCompleted" when in "Holding" state
/// Requires "Unhold" command to go to "Unholding" state 
{attribute 'object_name' := 'M_Held'}
METHOD M_Held
END_METHOD

/// Dynamic state "Holding"
/// Trigged by "Hold" command when in "Execute" state
/// Requires "StateCompleted" to go to "Held" state 
{attribute 'object_name' := 'M_Holding'}
METHOD M_Holding

 M_StateComplete();
END_METHOD

/// Static state "Idle"
/// Trigged by "StateCompleted" when in "Resetting" state
/// Requires "Start" command to go to "Starting" state 
{attribute 'object_name' := 'M_Idle'}
METHOD M_Idle
END_METHOD

METHOD PROTECTED M_Init : BOOL;
VAR_INPUT
END_VAR
IF NOT bInitDone THEN
	// Call method in base FB
	SUPER^.M_Init();

	bInitDone := TRUE;
END_IF
END_METHOD

METHOD M_JobDataHandling
VAR_INPUT
END_VAR
VAR
	sTempString : STRING(200);
END_VAR
// Job Data to device
IF (stJobDataIn.ChangeRequest <> stJobDataOut.ChangeStatus) AND (stJobDataIn.ChangeRequest > 0) THEN
	sTempString := CONCAT('NewJobdata request - Old request: ', TO_STRING(stJobDataOut.ChangeStatus));
	sTempString := CONCAT(sTempString, ', New request: ');
	sTempString := CONCAT(sTempString, TO_STRING(stJobDataIn.ChangeRequest));
	sTempString := CONCAT(sTempString, ' JobDataType: ');
	sTempString := CONCAT(sTempString, stJobDataIn.JobDataType); 	

	// Change request from Line Controller
	stJobDataOut.ChangeAcknowledge := stJobDataIn.ChangeRequest;
	
	

	// Check Job Type
	IF (stJobDataIn.JobDataType = 'OP11600') THEN	

		// Update output job data
		stJobDataOut.OP11600 := stJobDataIn.OP11600;
		stJobDataOut.JobDataType := stJobDataIn.JobDataType;

		// Signal that job data has been written		
		stJobDataOut.ChangeStatus := stJobDataIn.ChangeRequest;
		
		// Set job state to Idle
		stJobDataOut.JobState := 1;
		
		// Signal that output job data has been updated
		stJobDataOut.DataChange := stJobDataOut.DataChange + 1;

	ELSE

		// Update output job data
		stJobDataOut.JobDataType := '';

		// Signal that job data has been written		
		stJobDataOut.ChangeStatus := stJobDataIn.ChangeRequest;
		
		// Signal that output job data has been updated
		stJobDataOut.DataChange := stJobDataOut.DataChange + 1;

	END_IF
	
	sTempString := CONCAT(sTempString, ', TTarget: ');
	sTempString := CONCAT(sTempString, TO_STRING(stJobDataIn.OP11600.TemperatureTarget));
	sTempString := CONCAT(sTempString, ', TMin: ');
	sTempString := CONCAT(sTempString, TO_STRING(stJobDataIn.OP11600.TemperatureMin));
	sTempString := CONCAT(sTempString, ', TMax: ');
	sTempString := CONCAT(sTempString, TO_STRING(stJobDataIn.OP11600.TemperatureMax));
	sTempString := CONCAT(sTempString, ', SMin: ');
	sTempString := CONCAT(sTempString, TO_STRING(stJobDataIn.OP11600.SteamMin));
	sTempString := CONCAT(sTempString, ', SMax: ');
	sTempString := CONCAT(sTempString, TO_STRING(stJobDataIn.OP11600.SteamMax));
	sTempString := CONCAT(sTempString, ', AMin: ');
	sTempString := CONCAT(sTempString, TO_STRING(stJobDataIn.OP11600.AirMin));
	sTempString := CONCAT(sTempString, ', AMax: ');
	F_LogFile(CONCAT(sTempString, TO_STRING(stJobDataIn.OP11600.AirMax)));
END_IF
END_METHOD

/// Dynamic state "Resetting"
/// Trigged by "Reset" command when in "Stopped" state
/// Requires "StateCompleted" to go to "Idle" state 
{attribute 'object_name' := 'M_Resetting'}
METHOD M_Resetting
iOldChangeRequest := stJobDataIn.ChangeRequest;

M_StateComplete();
END_METHOD

/// Dynamic state "Starting"
/// Trigged by "Start" command when in "Idle" state
/// Requires "StateCompleted" to go to "Execute" state 
{attribute 'object_name' := 'M_Starting'}
METHOD M_Starting
// Starting production mode


// Start execute sequence

bStartLocal := FALSE;
eCommand := E_PML_Command.Undefined;


M_StateComplete();
END_METHOD

/// Static state "Stopped"
/// Trigged by "StateCompleted" when in "Stopping" state
/// Requires "Reset" command to go to "Resetting" state 
{attribute 'object_name' := 'M_Stopped'}
METHOD M_Stopped
END_METHOD

/// Dynamic state "Stopping"
/// Trigged by "Stop" command
/// Requires "StateCompleted" to go to "Stopped" state 
{attribute 'object_name' := 'M_Stopping'}
METHOD M_Stopping

 M_StateComplete();
END_METHOD

/// Static state "Suspended"
/// Trigged by "StateCompleted" when in "Suspending" state
/// Requires "Unsuspend" command to go to "Unsuspending" state 
{attribute 'object_name' := 'M_Suspended'}
METHOD M_Suspended
END_METHOD

/// Dynamic state "Suspending"
/// Trigged by "Suspend" command when in "Execute" state
/// Requires "StateCompleted" to go to "Suspended" state 
{attribute 'object_name' := 'M_Suspending'}
METHOD M_Suspending

 M_StateComplete();
END_METHOD

/// Dynamic state "Unholding"
/// Trigged by "Unhold" command when in "Held" state
/// Requires "StateCompleted" to go to "Execute" state 
{attribute 'object_name' := 'M_Unholding'}
METHOD M_Unholding

 M_StateComplete();
END_METHOD

/// Dynamic state "Unsuspending"
/// Trigged by "Unsuspend" command when in "Suspended" state
/// Requires "StateCompleted" to go to "Execute" state 
{attribute 'object_name' := 'M_Unsuspending'}
METHOD M_Unsuspending

 M_StateComplete();
END_METHOD

END_FUNCTION_BLOCK

// ---- ECC/TrackClient/FB_TrackClient.TcPOU
FUNCTION_BLOCK FB_TrackClient EXTENDS FB_TrackClient_Basic
VAR_INPUT
END_VAR
VAR_OUTPUT
END_VAR
VAR_IN_OUT
END_VAR
VAR
	// Station FB's
	afbStationCtrl			: ARRAY [1..5] OF FB_StationControl;
	
	// Decision Point
	eDecisionPointState		: E_DecisionPointState;
	nLastVehicleAtDecisionPoint: UINT;
	nLastVehicleAtStation1	: UINT;
	nLastVehicleAtStation2	: UINT;
	nLastPriorityInStation	: UINT;
	bDecisionPointBusy		: BOOL;
//	nDecisionPointVehicleNo	: UINT;
	nDecisionPointCellNo	: UINT;
	nDecisionPointBufferIdx	: USINT;
	sDecisionPointStationID	: STRING;
	tonDecisionPointDelay	: TON;
	bDecisionPoint_PAUSE	: BOOL;
	iDecisionPointMoveCmdID	: UINT;
	eDecisionPointMoveState	: E_VehicleMoveState;
	
	// Exit point
	eExitPointState			: E_ExitPointState;
	iExitPointStation		: UINT;
	iExitPointTicket		: UINT;
	iExitPointIndex			: UINT;
	iExitPointFirstIdx		: UINT;
	iExitPointBufferIdx		: UINT;
	tonExitPointDelay		: TON;
//	aExitPointVehicleNo		: ARRAY [1..MM_MAX_BUFFER_INDEX] OF UINT;	// Vehicle No's to be moved out by exit point logic
	iStation2MoveCmdID		: UINT;
	eStation2MoveState		: E_VehicleMoveState;
	arVehicleCommandBuffer	: ARRAY[0..10] OF ST_InputTransportCommand;
	bVehicleFoundCmdBuffer	: BOOL;
	bVehicleCmdPointer		: UINT;
	
	// Buffers handling
	ePostBufferIn			: E_PostBufferInState;
	ePostBufferOut			: E_PostBufferOutState;
	ePostBufferIn_Old		: E_PostBufferInState;
	ePostBufferOut_Old		: E_PostBufferOutState;
	eStationState			: E_StationState;
	eBufferStates			: E_BufferStates;
	eBufferState			: E_BufferState;
	iBufferStation			: UINT;
	iBufferTargetIDx		: USINT;
	iBufferSourceIDx		: UINT;
	tonBuffersDelay			: TON;
	iBufferMoveCmdID		: UINT;
	eBufferMoveState		: E_VehicleMoveState;
	afbBufferControlPre		: ARRAY[1..5] OF FB_BufferControl;
	afbBufferControlPost	: ARRAY[1..5] OF FB_BufferControl;
	
	// Vehicle FIFO (vehicles that are read from TrackServer but not belongs to this cell)
	aVehiclesStationFIFO	: ARRAY[1..10] OF ST_VehicleInHS;
	
	(* Misc *)
	stVehicleOnStation		: ST_ReadVehicleData;
	diBufferINStateTimer	: UINT;
	diBufferOUTStateTimer	: UINT;
	diStationStateTimer		: UINT;
	bBufferINStateChangeOS	: BOOL;
	bBufferOUTStateChangeOS	: BOOL;
	bStationStateChangeOS	: BOOL;
	eStationState_Old		: E_StationState;
	bStationEmpty			: BOOL;
	iVehicleFIFOOut			: UINT;
	bNextCell				: BOOL;
	bBufferFull				: BOOL;
	bVehicleAtStation		: BOOL;
	bIncludeStation			: BOOL;
	iVehicleCount			: UINT;
	iIDinx					: USINT;
	iIDoutx					: USINT;
	iBufferIdx				: UINT;
	iVehicleReadyStation1	: UINT;
	iVehicleReadyStation2	: UINT;
	iTicketToRemove			: UINT;
	iCurrentTicket			: UINT;
	iVehicleMoveBufferIN	: UINT;
	nVehicleNoToRemove		: UINT := 0;		// Vehicle number to remove from track system!
	bVehicleMovedFromSt1	: BOOL;

	iScanCnt: UINT;
	iNodeReads: UINT;
	iNodeReadErrs: UINT;
END_VAR

SUPER^(	stCommand := stCommand,
		stMappingIn := stMappingIn,
		stAdditionalDataIn := stAdditionalDataIn,
		stStatus := stStatus,
		stMappingOut := stMappingOut,
		stAdditionaldataOut := stAdditionaldataOut 	);

// Decision point
M_CTL_DecisionPoint();

// Exit point
//M_CTL_ExitPoint();

// Buffer handling
//M_CTL_Buffers();

// Station
M_CTL_Station();

METHOD M_ClearAll : BOOL
VAR_INPUT
END_VAR
VAR
	i	: UINT;
END_VAR
//Clear data on buffer locations
FOR i:=1 TO 5 DO
	IF aStations[i].bPresent THEN
		IF afbBufferControlPre[i].P_iBufferSize > 0 THEN
			afbBufferControlPre[i].M_ClearAll();
		END_IF
		IF afbBufferControlPost[i].P_iBufferSize > 0 THEN
			afbBufferControlPost[i].M_ClearAll();
		END_IF
	END_IF
END_FOR

//Clear data on station(s)
FOR i:=1 TO 5 DO
	IF aStations[i].bPresent THEN
		aStations[i].stStationData1.nTicket := 0;
		aStations[i].stStationData1.nTicketSize := 0;
		aStations[i].stStationData1.CurrentPriority := 0;
		aStations[i].stStationData1.nCurrentVehicleID := 0;
		aStations[i].stStationData1.nReservedVehicleID := 0;
		aStations[i].stStationData2.nTicket := 0;
		aStations[i].stStationData2.nTicketSize := 0;
		aStations[i].stStationData2.CurrentPriority := 0;
		aStations[i].stStationData2.nCurrentVehicleID := 0;
		aStations[i].stStationData2.nReservedVehicleID := 0;
	END_IF
END_FOR

//Clear statemachines
eBufferState := E_BufferState.Idle;
eExitPointState := E_ExitPointState.Idle;
eDecisionPointState := E_DecisionPointState.Idle;
//eMoveVehiclesOnCell := E_VehicleMoveState.Unknown;

////Clear various variables
bVehicleFoundCmdBuffer := FALSE;
MEMSET(ADR(arVehicleCommandBuffer), 0, SIZEOF(arVehicleCommandBuffer));
//bReadyStationIn[1] := FALSE;
//bReadyStationOut[1] := FALSE;
//bReadyStationOut[2] := FALSE;
//bST2OutVehicleOnTarget := FALSE;
//bST2InVehicleOnTarget := FALSE;
//bST1InVehicleOnTarget := FALSE;

//Clear StationControl
FOR i:= 1 TO 5 DO
	IF aStations[i].bPresent THEN
		afbStationCtrl[i].M_ClearAll();
		afbStationCtrl[i].bVehiclePreMoved := FALSE;
		afbStationCtrl[i].bVehiclePostMoved := FALSE;
		afbStationCtrl[i].bVehiclePreToInMoved := FALSE;
		afbStationCtrl[i].bVehiclePreToOutMoved := FALSE;
		afbStationCtrl[i].bVehicleInToOutMoved := FALSE;
		afbStationCtrl[i].bVehicleInToPostMoved := FALSE;
		afbStationCtrl[i].bVehicleOutToPostMoved := FALSE;
	END_IF
END_FOR

F_Logfile('TrackClient - All data cleared!');

M_ClearAll := TRUE;
END_METHOD

METHOD PROTECTED M_CommandData
VAR_INPUT
END_VAR
VAR
	i				: USINT;
	iRes			: UINT;
	bVehicleInCell	: BOOL;
END_VAR
// Handle the command data from OPC UA (stCommand)

// *** Speciel handling for this cell - addReservation have been moved to M_CTL_Station logic to delay until vehicle is fully complete ***

CASE eCommandDataState OF
	// Init state
	E_CommandDataState.Undefined:
		eCommandDataState := E_CommandDataState.CheckRequest;		

	// Check command data request
	E_CommandDataState.CheckRequest:
		IF ((stCommand.ChangeRequest <> stStatus.ChangeStatus) AND (stCommand.ChangeRequest > 0)) THEN
			// Check if changes is allowed on mapping data (from LC)
			IF (stAdditionalDataIn.MESHandShakes.DataChangeStatusTransportStatus = stStatus.DataChange) THEN
				stStatus.ChangeAcknowledge := stCommand.ChangeRequest;
				stStatus.DataChange := stStatus.DataChange + 1;
			
				// Find vehicle ID for specified Carrier ID
				iCommandDataVehicleID := M_CarrierIDToVehicleID(stCommand.CarrierID);
				IF ((iCommandDataVehicleID > 0) AND (iCommandDataVehicleID <= MM_MAX_NUMBER_OF_VEHICLE_ELEMENTS)) THEN
					// Specified vehicle found
					IF (F_StringCompNoCase(aReadVehicleData[iCommandDataVehicleID].stVehicle.sOwnerCell, sCellID)) THEN
						// Vehicle belongs to this cell
						stStatus.ValidRequest := TRUE;
						IF (stCommand.Ticket <= 0) THEN
							// Clear reservation data for this carrier (do not add reservation)
							eCommandDataState := E_CommandDataState.UpdateJobData;
						ELSE
							// Check if specified vehicle is inside this cell 
							bVehicleInCell := FALSE;
							FOR i := 1 TO 10 BY 1 DO
								IF F_StringCompNoCase(aVehiclesStationFIFO[i].sCarrierID, stCommand.CarrierID) THEN
									// Vehicle found
									bVehicleInCell := TRUE;
									EXIT;
								END_IF
							END_FOR
							IF (bVehicleInCell) THEN
								// Vehicle is currently being operated in this cell
								// Add reservation to buffer - to be send when ticket is complete
								FOR i := 0 TO 10 DO
									IF F_StringCompNoCase(arVehicleCommandBuffer[i].CarrierID, stCommand.CarrierID) THEN
										arVehicleCommandBuffer[i] := stCommand;
										F_LogLine(CONCAT('TC_CD: Command added to buffer (same), CarrierID: ', stCommand.CarrierID), 0);
										EXIT;
									ELSIF arVehicleCommandBuffer[i].CarrierID = '' THEN
										arVehicleCommandBuffer[i] := stCommand;
										F_LogLine(CONCAT('TC_CD: Command added to buffer (empty), CarrierID: ', stCommand.CarrierID), 0);
										EXIT;
									END_IF
								END_FOR
								eCommandDataState := E_CommandDataState.UpdateJobData;
							ELSE
								// Vehicle is NOT inside this cell
								// Add reservation to track server now
								F_LogLine(CONCAT('TC_CD: Handle command for CarrierID: ', stCommand.CarrierID), 0);
								eCommandDataState := E_CommandDataState.AddReservation;
							END_IF
						END_IF
					ELSE
						eCommandDataState := E_CommandDataState.Error;
					END_IF
				ELSE
					eCommandDataState := E_CommandDataState.Error;
				END_IF
			END_IF
		END_IF
		
	E_CommandDataState.AddReservation:
		iRes := M_CallAddReservation(	sStationID := stCommand.TargetStation,
										sCarrierID := stCommand.CarrierID,
										nTicket := stCommand.Ticket,
										nTicketSize := stCommand.CarriersInPackage,
										nPriority := stCommand.Priority 	);
		IF (iRes = 2) THEN
			// Success
			eCommandDataState := E_CommandDataState.UpdateJobData;
		ELSIF (iRes = 3) THEN
			// Error!
			eCommandDataState := E_CommandDataState.Error;
		END_IF
	
	E_CommandDataState.UpdateJobData:
		iRes := M_CallUpdateVehicleReservationData(	nVehicleID := iCommandDataVehicleID,
													sTargetStationID := stCommand.TargetStation,
													sCarrierID := stCommand.CarrierID,
													nTicket := stCommand.Ticket,
													nCarriersInPackage := stCommand.CarriersInPackage,
													nPriority := stCommand.Priority,
													sJobID := stCommand.JobID 	);
		IF (iRes = 2) THEN
			// Success
			eCommandDataState := E_CommandDataState.Done;
		ELSIF (iRes = 3) THEN
			// Error!
			eCommandDataState := E_CommandDataState.Error;
		END_IF
	
	E_CommandDataState.Done:
		stStatus.LatestTicket := stCommand.Ticket;
		stStatus.NumberOfCarriers := stCommand.CarriersInPackage;
		stStatus.ChangeStatus := stCommand.ChangeRequest;
		stStatus.DataChange := stStatus.DataChange + 1;
		eCommandDataState := E_CommandDataState.Undefined;
		
	E_CommandDataState.Error:
		stStatus.ValidRequest := FALSE;
		stStatus.ChangeStatus := stCommand.ChangeRequest;
		stStatus.DataChange := stStatus.DataChange + 1;
		eCommandDataState := E_CommandDataState.Undefined;
		
END_CASE
END_METHOD

METHOD PROTECTED M_CommandData_OLD
VAR_INPUT
END_VAR
VAR
	i			: USINT;
	iRes		: UINT;
END_VAR
// Handle the command data from OPC UA (stCommand)

// *** Speciel handling for this cell - addReservation have been moved to M_CTL_Station logic to delay until vehicle is fully complete ***

CASE eCommandDataState OF
	// Init state
	E_CommandDataState.Undefined:
		eCommandDataState := E_CommandDataState.CheckRequest;		

	// Check command data request
	E_CommandDataState.CheckRequest:
		IF ((stCommand.ChangeRequest <> stStatus.ChangeStatus) AND (stCommand.ChangeRequest > 0)) THEN
			// Check if changes is allowed on mapping data (from LC)
			IF (stAdditionalDataIn.MESHandShakes.DataChangeStatusTransportStatus = stStatus.DataChange) THEN
				stStatus.ChangeAcknowledge := stCommand.ChangeRequest;
				stStatus.DataChange := stStatus.DataChange + 1;
			
				// Find vehicle ID for specified Carrier ID
				iCommandDataVehicleID := M_CarrierIDToVehicleID(stCommand.CarrierID);
				IF ((iCommandDataVehicleID > 0) AND (iCommandDataVehicleID <= MM_MAX_NUMBER_OF_VEHICLE_ELEMENTS)) THEN
					// Specified vehicle found
					IF (F_StringCompNoCase(aReadVehicleData[iCommandDataVehicleID].stVehicle.sOwnerCell, sCellID)) THEN
						// Vehicle belongs to this cell
						stStatus.ValidRequest := TRUE;
						IF (stCommand.Ticket <= 0) THEN
							// Clear reservation data for this carrier (do not add reservation)
							eCommandDataState := E_CommandDataState.UpdateJobData;
						ELSE
//							// Add reservation to track server
//							eCommandDataState := E_CommandDataState.AddReservation;

							//Add reservation to buffer - to be send when ticket is complete
							FOR i := 0 TO 10 DO
								IF F_StringCompNoCase(arVehicleCommandBuffer[i].CarrierID, stCommand.CarrierID) THEN
									arVehicleCommandBuffer[i] := stCommand;
									F_LogLine('TC_CD: Command added to buffer same spot, VehicleID: %d', TO_UINT(stCommand.CarrierID));
									EXIT;
								ELSIF arVehicleCommandBuffer[i].CarrierID = '' THEN
									arVehicleCommandBuffer[i] := stCommand;
									F_LogLine('TC_CD: Command added to buffer empty spot, VehicleID: %d', TO_UINT(stCommand.CarrierID));
									EXIT;
								END_IF
							END_FOR
							eCommandDataState := E_CommandDataState.UpdateJobData;
						END_IF
					ELSE
						eCommandDataState := E_CommandDataState.Error;
					END_IF
				ELSE
					eCommandDataState := E_CommandDataState.Error;
				END_IF
			END_IF
		END_IF
		
	E_CommandDataState.AddReservation:
		iRes := M_CallAddReservation(	sStationID := stCommand.TargetStation,
										sCarrierID := stCommand.CarrierID,
										nTicket := stCommand.Ticket,
										nTicketSize := stCommand.CarriersInPackage,
										nPriority := stCommand.Priority 	);
		IF (iRes = 2) THEN
			// Success
			eCommandDataState := E_CommandDataState.UpdateJobData;
		ELSIF (iRes = 3) THEN
			// Error!
			eCommandDataState := E_CommandDataState.Error;
		END_IF
	
	E_CommandDataState.UpdateJobData:
		iRes := M_CallUpdateVehicleReservationData(	nVehicleID := iCommandDataVehicleID,
													sTargetStationID := stCommand.TargetStation,
													sCarrierID := stCommand.CarrierID,
													nTicket := stCommand.Ticket,
													nCarriersInPackage := stCommand.CarriersInPackage,
													nPriority := stCommand.Priority,
													sJobID := stCommand.JobID 	);
		IF (iRes = 2) THEN
			// Success
			eCommandDataState := E_CommandDataState.Done;
		ELSIF (iRes = 3) THEN
			// Error!
			eCommandDataState := E_CommandDataState.Error;
		END_IF
	
	E_CommandDataState.Done:
		stStatus.LatestTicket := stCommand.Ticket;
		stStatus.NumberOfCarriers := stCommand.CarriersInPackage;
		stStatus.ChangeStatus := stCommand.ChangeRequest;
		stStatus.DataChange := stStatus.DataChange + 1;
		eCommandDataState := E_CommandDataState.Undefined;
		
	E_CommandDataState.Error:
		stStatus.ValidRequest := FALSE;
		stStatus.ChangeStatus := stCommand.ChangeRequest;
		stStatus.DataChange := stStatus.DataChange + 1;
		eCommandDataState := E_CommandDataState.Undefined;
		
END_CASE
END_METHOD

METHOD M_CTL_Buffer : BOOL
VAR_INPUT
END_VAR
VAR
	iVehicleAtStation1 	: UINT;
	iVehicleAtStation2 	: UINT;
	iFirstStation		: UINT;
	i					: UINT;
	j					: UINT;
	iRes				: INT;
	sTempString			: STRING(200);

	bAllMoved			: BOOL;
END_VAR
iVehicleAtStation1 := M_CTL_VehicleAtStationX(iStationNo:= 1);
iVehicleAtStation2 := M_CTL_VehicleAtStationX(iStationNo:= 2);
//Run stateTimers
IF bBufferINStateChangeOS THEN
	diBufferInStateTimer := 0;
END_IF
IF diBufferInStateTimer < 64000 THEN
	diBufferInStateTimer := diBufferInStateTimer + g_iPLCScan_MS;
END_IF
IF bBufferOUTStateChangeOS THEN
	diBufferOutStateTimer := 0;
END_IF
IF diBufferOuTStateTimer < 64000 THEN
	diBufferOuTStateTimer := diBufferOUTStateTimer + g_iPLCScan_MS;
END_IF


//Get first station number
FOR i := 1 TO MM_MAX_NUMBER_OF_STATION_ELEMENTS DO
	IF NOT aReadStationData[i].stStationData.bStationPresent THEN EXIT; END_IF
	IF aReadStationData[i].stStationData.sCellID = 'C000004' THEN
		iFirstStation := i ;
		EXIT;
	END_IF
END_FOR


//Buffer IN
CASE ePostBufferIn OF
	E_PostBufferInState.Waiting:
	
		IF diBufferInStateTimer > 2000 AND NOT bBufferFull THEN
			//Vehicle FIFO out
//			IF LEN(aVehiclesStationFIFO[1].sCarrierID) > 0 THEN
//				IF aReadVehicleData[aVehiclesStationFIFO[1].nVehicleNo].stVehicle.sCurrentStationID = aStations[2].sStationID THEN
//					ePostBufferIn := E_PostBufferInState.FindPosition;
					
//					F_LogFile(CONCAT('BufferIN - FindPosition by first item in FIFO NO: ', TO_STRING(aVehiclesStationFIFO[1].nVehicleNo)));
//				END_IF
			//Vehicle at station
			IF iVehicleAtStation2 > 0 AND (nLastVehicleAtStation2 <> iVehicleAtStation2) THEN
				IF aStations[2].sStationID = aReadVehicleData[iVehicleAtStation2].stVehicle.sCurrentStationID THEN
					nLastVehicleAtStation2 := iVehicleAtStation2;
					ePostBufferIn := E_PostBufferInState.FindPosition;
					
					F_LogFile(CONCAT('BufferIN - FindPosition for vehicle at station NO: ', TO_STRING(iVehicleAtStation2)));
				END_IF 
			END_IF
			IF (iVehicleAtStation2 = 0) THEN
				// Previous vehicle removed from ST2. Reset Last vehicle ID (To allow same vehicle to arrive two times!)
				nLastVehicleAtStation2 := 0;
			END_IF
		END_IF
	
	E_PostBufferInState.FindPosition:
		IF ePostBufferOut = E_PostBufferOutState.CheckBuffer THEN
			FOR i := MM_MAX_BUFFER_INDEX TO 1 BY -1 DO
				IF aStations[2].astPostBuffer[i].bPresent AND aStations[2].astPostBuffer[i].nCurrentVehicleID = 0 THEN
					iIDinx := TO_USINT(i);
					ePostBufferIn := E_PostBufferInState.Infeed;
					
					iVehicleMoveBufferIN := iVehicleAtStation2;
					sTempString := CONCAT('BufferIN - Found pos at: ', TO_STRING(i));
					sTempString := CONCAT(sTempString, ', for vehicle NO: ');
					F_LogFile(CONCAT(sTempString, TO_STRING(iVehicleAtStation2)));
					EXIT;
				END_IF
			END_FOR
		
			//Looped through without finding a free position
			IF ePostBufferIn = E_PostBufferInState.FindPosition THEN
				aStations[2].stStationData1.nCurrentVehicleID := aReadStationData[iFirstStation+1].stStationData.nVehicleIDStationIn;
				aStations[2].stStationData1.nTicket := aReadVehicleData[iVehicleAtStation2].stVehicle.nTicket;
				aStations[2].stStationData1.nTicketSize := aReadVehicleData[iVehicleAtStation2].stVehicle.nTicketSize;
				bBufferFull := TRUE; (* Used in PostBufferOut *)
				nLastVehicleAtStation2 := 0; //Same vehicle for next check
				ePostBufferIn := E_PostBufferInState.Waiting;
				
				sTempString := ('BufferIN - Buffer full');
				F_LogFile(sTempString);
			ELSE
				bBufferFull := FALSE;
			END_IF
		END_IF
	E_PostBufferInState.Infeed:
		iRes := M_CallMoveVehicleToBuffer(	eInputType := E_MMVehicleInputType.eMMVehicleInputType_VehicleID, 
											sInput := UINT_TO_STRING(aReadStationData[iFirstStation+1].stStationData.nVehicleIDStationIn), 
											sStationID := afbStationCtrl[2].P_sStationID,
											eBufferType := E_MMStationBuffer.eMMStationBuffer_PostProcess, 
											nBufferIndex := iIDinx, 
											eDirection := E_MMDirection.eMMDirection_Forward, 
											fVelocity := 1, 
											fAcceleration := 1	);
		IF (iRes = 2) THEN
			// Movement call OK
			//Move data
			aStations[2].astPostBuffer[iIDinx].nCurrentVehicleID := aReadStationData[iFirstStation+1].stStationData.nVehicleIDStationIn;
			aStations[2].astPostBuffer[iIDinx].nTicket := aReadVehicleData[aStations[2].astPostBuffer[iIDinx].nCurrentVehicleID].stVehicle.nTicket;
			aStations[2].astPostBuffer[iIDinx].nTicketSize := aReadVehicleData[aStations[2].astPostBuffer[iIDinx].nCurrentVehicleID].stVehicle.nTicketSize;
			
			sTempString := CONCAT('BufferIN - Move to buffer OK NO: ', TO_STRING(aReadStationData[iFirstStation+1].stStationData.nVehicleIDStationIn));
			//Remove from FIFO
			IF LEN(aVehiclesStationFIFO[1].sCarrierID) > 0 THEN 
				IF nLastVehicleAtStation2 = aVehiclesStationFIFO[1].nVehicleNo THEN
					P_bFifoOut := TRUE;
					sTempString := CONCAT(sTempString, ', nLastVehicle: ');
					sTempString := CONCAT(sTempString, TO_STRING(nLastVehicleAtStation2));
					sTempString := CONCAT(sTempString, ', FIFO out carrierID: ');
					sTempString := CONCAT(sTempString, TO_STRING(aVehiclesStationFIFO[1].nVehicleNo));
//					sTempString := CONCAT(sTempString, ' Removed from FIFO');
					
//					aVehiclesStationFIFO[1].nVehicleNo := 0;
//					aVehiclesStationFIFO[1].sCarrierID := '';
	
				END_IF
			END_IF
			F_LogFile(sTempString);
			ePostBufferIn := E_PostBufferInState.ExtraVehicleRemove;
			
		ELSIF (iRes = 3) THEN
			// Movement call failed
			// TODO!!!
			F_LogFile(CONCAT('BufferIN - Move to buffer FAILED NO: ', TO_STRING(aReadStationData[iFirstStation+1].stStationData.nVehicleIDStationIn)));
			ePostBufferIn := E_PostBufferInState.ExtraVehicleRemove;

		END_IF
		
	E_PostBufferInState.ExtraVehicleRemove:
(*	Wait ro remove until moved out from post buffer!
		IF M_ExtraVehicleRemove(iVehicleNo:= iVehicleMoveBufferIN) THEN
			F_LogFile(CONCAT('BufferIN - Vehicle removed from extra, NO: ', TO_STRING(aReadStationData[iFirstStation+1].stStationData.nVehicleIDStationIn)));
			ePostBufferIn := E_PostBufferInState.Waiting;
		END_IF
*)
		ePostBufferIn := E_PostBufferInState.Waiting;

END_CASE


//Buffer out
CASE ePostBufferOut OF
	E_PostBufferOutState.Waiting:
		tonPostBufferDelay.IN := FALSE;
		FOR i := 1 TO MM_MAX_BUFFER_INDEX BY 1 DO
			aPostBufferVehicleNo[i] := 0;
		END_FOR
		ePostBufferOut := E_PostBufferOutState.CheckBufferSpace;
		F_LogFile('BufferOUT - Waiting -> CheckBufferSpace');
		
	E_PostBufferOutState.CheckBuffer:
		iVehicleCount := 0;
		bIncludeStation := FALSE;
		//Loop through buffers and check tickets
		FOR i := MM_MAX_BUFFER_INDEX TO 1 BY -1 DO
			IF aStations[2].astPostBuffer[i].bPresent AND aStations[2].astPostBuffer[i].nCurrentVehicleID <> 0 THEN
				iVehicleCount := iVehicleCount +1;
				
				//Ticket number differs	- send out vehicles
				IF iVehicleCount > 1 AND (aStations[2].astPostBuffer[i+1].nTicket <> aStations[2].astPostBuffer[i].nTicket) THEN
					iVehicleCount := iVehicleCount - 1;
					ePostBufferOut := E_PostBufferOutState.SetTrafficLightRed;
		
					sTempString := CONCAT('BufferOUT - Diff ticket, found: ', TO_STRING(iVehicleCount+1));
					sTempString := CONCAT(sTempString, ', of vehicle(s), old ticket: ');
					sTempString := CONCAT(sTempString, TO_STRING(aStations[2].astPostBuffer[i+1].nTicket));
					sTempString := CONCAT(sTempString, ', new ticket: ');
					F_LogFile(CONCAT(sTempString, TO_STRING(aStations[2].astPostBuffer[i].nTicket)));
					EXIT;
				//Vehicle count with amount of tickets reached
				ELSIF iVehicleCount > 0 AND (iVehicleCount >= aStations[2].astPostBuffer[i].nTicketSize OR aStations[2].astPostBuffer[i].nTicket = 0) THEN
					ePostBufferOut := E_PostBufferOutState.SetTrafficLightRed;
					
					sTempString := CONCAT('BufferOUT - All tickets found or ticket = 0: ', TO_STRING(iVehicleCount));
					sTempString := CONCAT(sTempString, ', of vehicle(s), ticket: ');
					sTempString := CONCAT(sTempString, TO_STRING(aStations[2].astPostBuffer[i].nTicket));
					sTempString := CONCAT(sTempString, ', of ticket size: ');
					F_LogFile(CONCAT(sTempString, TO_STRING(aStations[2].astPostBuffer[i].nTicketSize)));		
					EXIT;
				END_IF
			END_IF
		END_FOR
		//Buffer full check with vehicle on station
		IF bBufferFull AND iVehicleCount > 1 THEN
			//Ticket number differs	- send out vehicles
			IF (aStations[2].stStationData1.nTicket <> aStations[2].astPostBuffer[1].nTicket) THEN
				ePostBufferOut := E_PostBufferOutState.SetTrafficLightRed;
				
				sTempString := CONCAT('BufferOUT - Diff ticket, buffer full found: ', TO_STRING(iVehicleCount));
				sTempString := CONCAT(sTempString, ', of vehicle(s), ticket on station: ');
				sTempString := CONCAT(sTempString, TO_STRING(aStations[2].stStationData1.nTicket));
				sTempString := CONCAT(sTempString, ', ticket on pos 1 buffer: ');
				F_LogFile(CONCAT(sTempString, TO_STRING(aStations[2].astPostBuffer[1].nTicket)));
			//Vehicle count with amount of tickets reached
			ELSE 
				bIncludeStation := TRUE;
				nLastVehicleAtStation2 := iVehicleAtStation2;
				ePostBufferOut := E_PostBufferOutState.SetTrafficLightRed;

				sTempString := CONCAT('BufferOUT - Buffer full found: ', TO_STRING(iVehicleCount));
				sTempString := CONCAT(sTempString, ', of vehicle(s), ticket on station: ');
				sTempString := CONCAT(sTempString, TO_STRING(aStations[2].stStationData1.nTicket));
				sTempString := CONCAT(sTempString, ', ticket on pos 1 buffer: ');
				F_LogFile(CONCAT(sTempString, TO_STRING(aStations[2].astPostBuffer[1].nTicket)));		
			END_IF
		END_IF
		
		iBufferIdx := MM_MAX_BUFFER_INDEX;
		iIDoutx := TO_USINT(iVehicleCount);
	
	E_PostBufferOutState.SetTrafficLightRed:
		IF diBufferOUTStateTimer > 2000 THEN
			iRes := M_CallSetTrafficLightColor(	nColor := E_MMTrafficLightColor.eMMTrafficLightColor_Red );
			IF (iRes = 2) THEN
				// Call OK
				ePostBufferOut := E_PostBufferOutState.Outfeed;
				F_LogFile('BufferOUT - Set trafficlight RED OK');
			ELSIF (iRes = 3) THEN
				// Call failed
				// TODO!!!
				ePostBufferOut := E_PostBufferOutState.Waiting;
				F_LogFile('BufferOUT - Set trafficlight FAILED');
			END_IF
		END_IF
		
	E_PostBufferOutState.Outfeed:
		IF diBufferOUTStateTimer > 2000 THEN
			IF aStations[2].astPostBuffer[iBufferIdx].bPresent THEN
				iRes := M_CallMoveVehicleToDecisionPoint(eInputType := E_MMVehicleInputType.eMMVehicleInputType_VehicleID, 
														 sInput := UINT_TO_STRING(aStations[2].astPostBuffer[iBufferIdx].nCurrentVehicleID), 
														 sStationID := sNextStationOnTrack,
														 eDirection := E_MMDirection.eMMDirection_Forward, 
														 fVelocity := 1, 
														 fAcceleration := 1	);
				IF (iRes = 2) THEN
					// Movement call OK
					sTempString := CONCAT('BufferOUT - Move vehicle: ', TO_STRING(aStations[2].astPostBuffer[iBufferIdx].nCurrentVehicleID));
					F_LogFile(CONCAT(sTempString, ', out OK'));
					// Save vehicle numbers for moved vehicles
					aPostBufferVehicleNo[iBufferIdx] := aStations[2].astPostBuffer[iBufferIdx].nCurrentVehicleID;
					// Clear buffer data					
					aStations[2].astPostBuffer[iBufferIdx].nCurrentVehicleID := 0;
					aStations[2].astPostBuffer[iBufferIdx].nTicket := 0;
					aStations[2].astPostBuffer[iBufferIdx].nTicketSize := 0;
					iBufferIdx := iBufferIdx - 1;
					iIDoutx := iIDoutx -1;
		
					IF (iIDoutx <= 0) THEN
						// All in buffer move - move on station?
						IF bIncludeStation THEN
							ePostBufferOut := E_PostBufferOutState.OutfeedStation;
							bBufferFull := FALSE;
							F_LogFile('BufferOUT - include station');
						ELSE
							ePostBufferOut := E_PostBufferOutState.WaitOutfeedStation;
							
							F_LogFile('BufferOUT - NOT include station');
						END_IF	
					END_IF
				ELSIF (iRes = 3) THEN
					// Movement call failed
					// TODO!!!
				END_IF
			ELSE
				iBufferIdx := LIMIT(1, (iBufferIdx - 1), MM_MAX_BUFFER_INDEX);
			END_IF
		END_IF
	
	E_PostBufferOutState.OutfeedStation:
		iRes := M_CallMoveVehicleToDecisionPoint(eInputType := E_MMVehicleInputType.eMMVehicleInputType_VehicleID, 
														 sInput := UINT_TO_STRING(aStations[2].stStationData1.nCurrentVehicleID), 
														 sStationID := sNextStationOnTrack,
														 eDirection := E_MMDirection.eMMDirection_Forward, 
														 fVelocity := 1, 
														 fAcceleration := 1	);
		IF (iRes = 2) THEN
			// Movement call OK
			// Save vehicle numbers for moved vehicles (use index 0 for buffer position)
			aPostBufferVehicleNo[0] := aStations[2].stStationData1.nCurrentVehicleID;
			// Clear buffer data					
			aStations[2].stStationData1.nCurrentVehicleID := 0;
			aStations[2].stStationData1.nTicket := 0;
			aStations[2].stStationData1.nTicketSize := 0;
			ePostBufferOut := E_PostBufferOutState.WaitOutfeedStation;
			F_LogFile('BufferOUT - Move to station OK');
		ELSIF (iRes = 3) THEN
			// Movement call failed
			// TODO!!!
		END_IF
	
// TEST
	E_PostBufferOutState.WaitOutfeedStation:
		tonPostBufferDelay.IN := TRUE;
		tonPostBufferDelay.PT := T#60S;
		IF ((tonPostBufferDelay.ET > T#4S)) THEN
			bAllMoved := TRUE;
			// Check if all vehicles are moved away from station path ID
			FOR i := 0 TO MM_MAX_BUFFER_INDEX BY 1 DO
				IF (aPostBufferVehicleNo[i] > 0) THEN
					// Vehicle no to be checked!
					IF (aReadVehicleData[aPostBufferVehicleNo[i]].stVehicle.nPathID <> aStations[2].stStationData1.stLocation.nPathID) THEN
						// This vehicle IS away from station path
						// Stop checking it
						M_ExtraVehicleRemove(iVehicleNo:= aPostBufferVehicleNo[i]);
						F_LogFile(CONCAT('BufferOUT - Move to station DONE. NO: ', UINT_TO_STRING(aPostBufferVehicleNo[i])));
						aPostBufferVehicleNo[i] := 0;
					ELSE
						// This vehicle is NOT away from station path
						bAllMoved := FALSE;
						EXIT;
					END_IF
				END_IF
			END_FOR
			IF (bAllMoved OR tonPostBufferDelay.Q) THEN
				tonPostBufferDelay.IN := FALSE;
				ePostBufferOut := E_PostBufferOutState.SetTrafficLightGreen;			
			END_IF
		END_IF
// TEST END 
		
	E_PostBufferOutState.SetTrafficLightGreen:
		IF diBufferOutStateTimer > 3000 THEN
			iRes := M_CallSetTrafficLightColor(	nColor := E_MMTrafficLightColor.eMMTrafficLightColor_Green );
			IF (iRes = 2) THEN
				// Call OK
				bBufferFull := FALSE;
				ePostBufferOut := E_PostBufferOutState.CheckBufferSpace;
				F_LogFile('BufferOUT - Traffic light green OK');
			ELSIF (iRes = 3) THEN
				bBufferFull := FALSE;
				// Call failed
				F_LogFile('BufferOUT - Traffic light green Failed!');
				// TODO!!!
				ePostBufferOut := E_PostBufferOutState.CheckBufferSpace;
			END_IF
		END_IF

	E_PostBufferOutState.CheckBufferSpace:
		IF diBufferOutStateTimer > 2000 THEN
			FOR i := MM_MAX_BUFFER_INDEX TO 1 BY -1 DO
				IF i > 1 AND
					aStations[2].astPostBuffer[i].bPresent AND aStations[2].astPostBuffer[i].nCurrentVehicleID = 0 AND
					aStations[2].astPostBuffer[i-1].nCurrentVehicleID <> 0 THEN
					ePostBufferOut := E_PostBufferOutState.Acumulate;
					iIDoutx := TO_USINT(i);
					
					sTempString := CONCAT('BufferOUT - Accumulate, move vehicle: ', TO_STRING(aStations[2].astPostBuffer[i-1].nCurrentVehicleID));
					sTempString := CONCAT(sTempString, ', From buffer pos: ');
					sTempString := CONCAT(sTempString, TO_STRING(i-1));
					sTempString := CONCAT(sTempString, ', to buffer pos: ');
					sTempString := CONCAT(sTempString, TO_STRING(i));
					sTempString := CONCAT(sTempString, ', for station: ');
					F_LogFile(CONCAT(sTempString, afbStationCtrl[2].P_sStationID));		
					EXIT;
				
				ELSIF i <= 1 THEN
					ePostBufferOut := E_PostBufferOutState.CheckBuffer;
					F_LogFile('BufferOUT - Check buffer space DONE');
					EXIT;
				END_IF
			END_FOR
		END_IF
				
	E_PostBufferOutState.Acumulate:
		iRes := M_CallMoveVehicleToBuffer(	eInputType := E_MMVehicleInputType.eMMVehicleInputType_VehicleID, 
											sInput := UINT_TO_STRING(aStations[2].astPostBuffer[iIDoutX-1].nCurrentVehicleID), 
											sStationID := afbStationCtrl[2].P_sStationID,
											eBufferType := E_MMStationBuffer.eMMStationBuffer_PostProcess, 
											nBufferIndex := iIDoutx, 
											eDirection := E_MMDirection.eMMDirection_Forward, 
											fVelocity := 1, 
											fAcceleration := 1	);

		IF (iRes = 2) THEN
			// Movement call OK
			//Move data
			M_CopyAndClearBufferData(stSource:= aStations[2].astPostBuffer[iIDoutx-1], stTarget:= aStations[2].astPostBuffer[iIDoutx]);
			bBufferFull := FALSE;
			ePostBufferOut := E_PostBufferOutState.CheckBufferSpace;
			F_LogFile('BufferOUT - Acummulate OK');
		ELSIF (iRes = 3) THEN
			// Movement call failed
			// TODO!!!
			bBufferFull := FALSE;
			ePostBufferOut := E_PostBufferOutState.Waiting;
			F_LogFile('BufferOUT - Acummulate FAILED');
		END_IF
END_CASE


//OS state Change
bBufferINStateChangeOS := ePostBufferIn <> ePostBufferIn_Old;
ePostBufferIn_Old := ePostBufferIn;

bBufferOUTStateChangeOS := ePostBufferOut <> ePostBufferOut_Old;
ePostBufferOut_Old := ePostBufferOut;

// Delay
tonPostBufferDelay(	IN:= ,
					PT:= ,
					Q=> ,
					ET=> 	);
END_METHOD

/// Handle buffers
METHOD PROTECTED M_CTL_Buffers
VAR_INPUT
END_VAR
VAR
	iRes				: INT;
END_VAR

CASE eBufferState OF
	E_BufferState.Idle:
		tonBuffersDelay.IN := FALSE;
		IF (bEnable AND bConnectedMethod AND bConnectedNode) THEN
			eBufferState := E_BufferState.Waiting;
		ELSE
			iBufferStation := 1;
		END_IF
		
	E_BufferState.Waiting:
		//IF ((eDecisionPointState = E_DecisionPointState.Idle) OR (eDecisionPointState = E_DecisionPointState.WaitStationEmpty) OR (eDecisionPointState = E_DecisionPointState.WaitStationReady)) THEN
			// Buffers can be handled now
			eBufferState := E_BufferState.CheckBuffer;
		//END_IF
		
	E_BufferState.CheckBuffer:
		IF (afbStationCtrl[iBufferStation].bMoveVehiclePreToIn) THEN
			// Station control request a vehicle move from pre buffer to station input location
			eBufferState := E_BufferState.WaitPreToInOnPos;			
		ELSIF (afbStationCtrl[iBufferStation].bMoveVehiclePreToOut) THEN
			// Station control request a vehicle move from pre buffer to station output location
			eBufferState := E_BufferState.WaitPreToOutOnPos;			
		ELSIF (afbStationCtrl[iBufferStation].bMoveVehicleInToOut) THEN
			// Station control request a vehicle move from station input to station output
			eBufferState := E_BufferState.MoveInToOut;			
		ELSIF (afbStationCtrl[iBufferStation].bMoveVehicleOutToPost) THEN
			// Station control request a vehicle move from station output to post buffer
			eBufferState := E_BufferState.MoveOutToPost;			
		ELSIF (afbStationCtrl[iBufferStation].bMoveVehicleInToPost) THEN
			// Station control request a vehicle move from station input to post buffer
			eBufferState := E_BufferState.MoveInToPost;
		ELSE
			iBufferStation := iBufferStation + 1;
			IF ( (iBufferStation > 5) OR (NOT aStations[iBufferStation].bPresent) ) THEN
				// Start from beginning
				iBufferStation := 1;
			END_IF
			eBufferState := E_BufferState.Idle;			
		END_IF

/////////////////////////////////////////////////////////////////////////////////////////////////////////////////////////////////////////////////////////
// Station input/pickup
/////////////////////////////////////////////////////////////////////////////////////////////////////////////////////////////////////////////////////////	
	E_BufferState.WaitPreToInOnPos:
		tonBuffersDelay.IN := TRUE;
		tonBuffersDelay.PT := T#0S;
		IF (tonBuffersDelay.Q) THEN
			iRes := M_CallMoveVehicleStatus(iCommandID := afbBufferControlPre[1].P_iCurrentVehicleCmdID,
												eMoveStatus => eBufferMoveState 	);
			
				IF (iRes = 2) THEN
					tonBuffersDelay.IN := FALSE;
					// Call OK
					IF (eBufferMoveState >= E_VehicleMoveState.ErrorLocation) THEN
						// Error with command
						// TODO!!!
						
					ELSIF (eBufferMoveState >= E_VehicleMoveState.Complete) THEN
						// Command accepted!
						F_LogLine('TC_BUF: Pre-Buf Vehicle on Pos : %d', afbBufferControlPre[1].P_iCurrentVehicleID);
						eBufferState := E_BufferState.MovePreToIn;
					END_IF
					
				ELSIF (iRes = 3) THEN
					tonBuffersDelay.IN := FALSE;
				// Movement call failed... Retry
				
				END_IF
			END_IF
	
	E_BufferState.MovePreToIn:
		iRes := M_CallMoveVehicleToStationIn(	eInputType := E_MMVehicleInputType.eMMVehicleInputType_VehicleID, 
												sInput := UINT_TO_STRING(aStations[iBufferStation].astPreBuffer[1].nCurrentVehicleID), 
												sStationID := afbStationCtrl[iBufferStation].P_sStationID,
												eDirection := E_MMDirection.eMMDirection_Forward, 
												fVelocity := 0.5, 
												fAcceleration := 1,
												iCmdID => iBufferMoveCmdID 	);
		IF (iRes = 2) THEN
			// Movement call OK
			// Trig event-driven reading
			M_VehicleToReadAdd(aStations[iBufferStation].astPreBuffer[1].nCurrentVehicleID);
			F_LogLine('TC_BUF: Pre-Buf To In OK : %d', aStations[iBufferStation].astPreBuffer[1].nCurrentVehicleID);				
			eBufferState := E_BufferState.WaitPreToIn;
		ELSIF (iRes = 3) THEN
			// Movement call failed
			// TODO!!!
			F_LogLine('TC_BUF: Error moving Pre-Buf To In! : %d', aStations[iBufferStation].astPreBuffer[1].nCurrentVehicleID);
			eBufferState := E_BufferState.Idle;
		END_IF
	
	E_BufferState.WaitPreToIn:
		tonBuffersDelay.IN := TRUE;
		tonBuffersDelay.PT := T#1S;
		IF (tonBuffersDelay.Q) THEN
			iRes := M_CallMoveVehicleStatus(iCommandID := iBufferMoveCmdID,
											eMoveStatus => eBufferMoveState 	);
			IF (iRes = 2) THEN
				tonBuffersDelay.IN := FALSE;
				// Call OK
				IF (eBufferMoveState >= E_VehicleMoveState.ErrorLocation) THEN
					// Error with command
					// TODO!!!
					
				ELSIF (eBufferMoveState = E_VehicleMoveState.Complete) THEN
					// Command completed!
					// Trig event-driven reading
					M_VehicleToReadAdd(aStations[iBufferStation].astPreBuffer[1].nCurrentVehicleID);			
					// Update buffer data			
					M_CopyBufferData(stSource := aStations[iBufferStation].astPreBuffer[1], stTarget := aStations[iBufferStation].stStationData1);
					//Delete from buffercontrol
					afbBufferControlPre[iBufferStation].M_RemoveVehicle(iVehicleID:= aStations[iBufferStation].astPreBuffer[1].nCurrentVehicleID);
					// signal movement finished
					afbStationCtrl[iBufferStation].bVehiclePreToInMoved := TRUE;
					eBufferState := E_BufferState.FinishedPreToIn;
					
				END_IF
				
			ELSIF (iRes = 3) THEN
				tonBuffersDelay.IN := FALSE;
				// Movement call failed... Retry
				
			END_IF
		END_IF

	E_BufferState.FinishedPreToIn:
		IF (NOT afbStationCtrl[iBufferStation].bMoveVehiclePreToIn) THEN
			afbStationCtrl[iBufferStation].bVehiclePreToInMoved := FALSE;
			eBufferState := E_BufferState.Idle;
		END_IF

/////////////////////////////////////////////////////////////////////////////////////////////////////////////////////////////////////////////////////////
// Station output/place
/////////////////////////////////////////////////////////////////////////////////////////////////////////////////////////////////////////////////////////
	E_BufferState.WaitPreToOutOnPos:
		tonBuffersDelay.IN := TRUE;
		tonBuffersDelay.PT := T#0S;
		IF (tonBuffersDelay.Q) THEN
			iRes := M_CallMoveVehicleStatus(iCommandID := afbBufferControlPre[1].P_iCurrentVehicleCmdID,
												eMoveStatus => eBufferMoveState 	);
			
				IF (iRes = 2) THEN
					tonBuffersDelay.IN := FALSE;
					// Call OK
					IF (eBufferMoveState >= E_VehicleMoveState.ErrorLocation) THEN
						// Error with command
						// TODO!!!
						
					ELSIF (eBufferMoveState >= E_VehicleMoveState.Complete) THEN
						// Command accepted!
						F_LogLine('TC_BUF: Pre-Buf Vehicle on Pos : %d', afbBufferControlPre[1].P_iCurrentVehicleID);
						eBufferState := E_BufferState.MovePreToOut;
					END_IF
					
				ELSIF (iRes = 3) THEN
					tonBuffersDelay.IN := FALSE;
				// Movement call failed... Retry
				
				END_IF
			END_IF

	E_BufferState.MovePreToOut:
		iRes := M_CallMoveVehicleToStationOut(	eInputType := E_MMVehicleInputType.eMMVehicleInputType_VehicleID, 
												sInput := UINT_TO_STRING(aStations[iBufferStation].astPreBuffer[1].nCurrentVehicleID), 
												sStationID := afbStationCtrl[iBufferStation].P_sStationID,
												eDirection := E_MMDirection.eMMDirection_Forward, 
												fVelocity := 0.5, 
												fAcceleration := 1,
												iCmdID => iBufferMoveCmdID 	);
		IF (iRes = 2) THEN
			// Movement call OK
			// Trig event-driven reading
			M_VehicleToReadAdd(aStations[iBufferStation].astPreBuffer[1].nCurrentVehicleID);
			F_LogLine('TC_BUF: Moving Pre-Buf To Out OK : %d', aStations[iBufferStation].astPreBuffer[1].nCurrentVehicleID);				
			eBufferState := E_BufferState.WaitPreToOut;
		ELSIF (iRes = 3) THEN
			// Movement call failed
			// TODO!!!
			F_LogLine('TC_BUF: Error moving Pre-Buf To Out! : %d', aStations[iBufferStation].astPreBuffer[1].nCurrentVehicleID);
			eBufferState := E_BufferState.Idle;
		END_IF
	
	E_BufferState.WaitPreToOut:
		tonBuffersDelay.IN := TRUE;
		tonBuffersDelay.PT := T#1S;
		IF (tonBuffersDelay.Q) THEN
			iRes := M_CallMoveVehicleStatus(iCommandID := iBufferMoveCmdID,
											eMoveStatus => eBufferMoveState 	);
			IF (iRes = 2) THEN
				tonBuffersDelay.IN := FALSE;
				// Call OK
				IF (eBufferMoveState >= E_VehicleMoveState.ErrorLocation) THEN
					// Error with command
					// TODO!!!
					
				ELSIF (eBufferMoveState = E_VehicleMoveState.Complete) THEN
					// Command completed!
					// Trig event-driven reading
					M_VehicleToReadAdd(aStations[iBufferStation].astPreBuffer[1].nCurrentVehicleID);				
					// Update buffer data			
					M_CopyBufferData(stSource := aStations[iBufferStation].astPreBuffer[1], stTarget := aStations[iBufferStation].stStationData2);
					//Delete from buffercontrol
					afbBufferControlPre[iBufferStation].M_RemoveVehicle(iVehicleID:= aStations[iBufferStation].astPreBuffer[1].nCurrentVehicleID);
					// signal movement finished
					afbStationCtrl[iBufferStation].bVehiclePreToOutMoved := TRUE;
					eBufferState := E_BufferState.FinishedPreToOut;
					
				END_IF
				
			ELSIF (iRes = 3) THEN
				tonBuffersDelay.IN := FALSE;
				// Movement call failed... Retry
				
			END_IF
		END_IF

	E_BufferState.FinishedPreToOut:
		IF (NOT afbStationCtrl[iBufferStation].bMoveVehiclePreToOut) THEN
			afbStationCtrl[iBufferStation].bVehiclePreToOutMoved := FALSE;
			eBufferState := E_BufferState.Idle;
		END_IF

/////////////////////////////////////////////////////////////////////////////////////////////////////////////////////////////////////////////////////////
// Station input to Station output
/////////////////////////////////////////////////////////////////////////////////////////////////////////////////////////////////////////////////////////		
	E_BufferState.MoveInToOut:
	// TODO!!! - Vehicle ID of vehicle in station IN location?
		iRes := M_CallMoveVehicleToStationOut(	eInputType := E_MMVehicleInputType.eMMVehicleInputType_VehicleID, 
												sInput := UINT_TO_STRING(aStations[iBufferStation].stStationData1.nCurrentVehicleID), 
												sStationID := afbStationCtrl[iBufferStation].P_sStationID,
												eDirection := E_MMDirection.eMMDirection_Forward, 
												fVelocity := 0.5, 
												fAcceleration := 1,
												iCmdID => iBufferMoveCmdID 	);
		IF (iRes = 2) THEN
			// Movement call OK
			// Trig event-driven reading
			M_VehicleToReadAdd(aStations[iBufferStation].stStationData1.nCurrentVehicleID);		
			F_LogLine('TC_BUF: Moving In To Out OK : %d', aStations[iBufferStation].stStationData1.nCurrentVehicleID);			
			eBufferState := E_BufferState.WaitInToOut;
		ELSIF (iRes = 3) THEN
			// Movement call failed
			// TODO!!!
			F_LogLine('TC_BUF: Error moving In To Out! : %d', aStations[iBufferStation].stStationData1.nCurrentVehicleID);
			eBufferState := E_BufferState.Idle;
		END_IF
	
	E_BufferState.WaitInToOut:
		tonBuffersDelay.IN := TRUE;
		tonBuffersDelay.PT := T#1S;
		IF (tonBuffersDelay.Q) THEN
			iRes := M_CallMoveVehicleStatus(iCommandID := iBufferMoveCmdID,
											eMoveStatus => eBufferMoveState 	);
			IF (iRes = 2) THEN
				tonBuffersDelay.IN := FALSE;
				// Call OK
				IF (eBufferMoveState >= E_VehicleMoveState.ErrorLocation) THEN
					// Error with command
					// TODO!!!
					
				ELSIF (eBufferMoveState = E_VehicleMoveState.Complete) THEN
					// Command completed!
					// Trig event-driven reading
					M_VehicleToReadAdd(aStations[iBufferStation].stStationData1.nCurrentVehicleID);				
					// Update buffer data			
					M_CopyAndClearBufferData(stSource := aStations[iBufferStation].stStationData1, stTarget := aStations[iBufferStation].stStationData2);
					// signal movement finished
					afbStationCtrl[iBufferStation].bVehicleInToOutMoved := TRUE;
					eBufferState := E_BufferState.FinishedInToOut;
					
				END_IF
				
			ELSIF (iRes = 3) THEN
				tonBuffersDelay.IN := FALSE;
				// Movement call failed... Retry
				
			END_IF
		END_IF

	E_BufferState.FinishedInToOut:
		IF (NOT afbStationCtrl[iBufferStation].bMoveVehicleInToOut) THEN
			afbStationCtrl[iBufferStation].bVehicleInToOutMoved := FALSE;
			eBufferState := E_BufferState.Idle;
		END_IF

/////////////////////////////////////////////////////////////////////////////////////////////////////////////////////////////////////////////////////////
// Station output to post buffer
/////////////////////////////////////////////////////////////////////////////////////////////////////////////////////////////////////////////////////////		
	E_BufferState.MoveOutToPost:
	// TODO!!! - Vehicle ID of vehicle in station OUT location?
		iRes := M_CallMoveVehicleToBuffer(	eInputType := E_MMVehicleInputType.eMMVehicleInputType_VehicleID, 
											sInput := UINT_TO_STRING(aStations[iBufferStation].stStationData2.nCurrentVehicleID), 
											sStationID := afbStationCtrl[iBufferStation].P_sStationID,
											eBufferType := E_MMStationBuffer.eMMStationBuffer_PostProcess, 
											nBufferIndex := TO_USINT(afbBufferControlPost[iBufferStation].P_iBufferSize), // Last location in buffer 
											eDirection := E_MMDirection.eMMDirection_Forward, 
											fVelocity := 0.5, 
											fAcceleration := 1,
											iCmdID => iBufferMoveCmdID 	);
		IF (iRes = 2) THEN
			// Movement call OK
			// Trig event-driven reading
			M_VehicleToReadAdd(aStations[iBufferStation].stStationData2.nCurrentVehicleID);				
			eBufferState := E_BufferState.WaitOutToPost;
		ELSIF (iRes = 3) THEN
			// Movement call failed
			// TODO!!!
			F_LogLine('TC_BUF: Error moving Out To Post-Buf! : %d', aStations[iBufferStation].stStationData2.nCurrentVehicleID);
			eBufferState := E_BufferState.Idle;
		END_IF
	
	E_BufferState.WaitOutToPost:
		tonBuffersDelay.IN := TRUE;
		tonBuffersDelay.PT := T#500MS;
		IF (tonBuffersDelay.Q) THEN
			iRes := M_CallMoveVehicleStatus(iCommandID := iBufferMoveCmdID,
											eMoveStatus => eBufferMoveState 	);
			IF (iRes = 2) THEN
				tonBuffersDelay.IN := FALSE;
				// Call OK
				IF (eBufferMoveState >= E_VehicleMoveState.ErrorLocation) THEN
					// Error with command
					// TODO!!!
					
				ELSIF (eBufferMoveState = E_VehicleMoveState.Moving OR eBufferMoveState = E_VehicleMoveState.Complete) THEN
					// Command completed!
					// Trig event-driven reading
					M_VehicleToReadAdd(aStations[iBufferStation].stStationData2.nCurrentVehicleID);				
		
					// Check if ticket size in 1 
					IF (aStations[1].stStationData2.nTicketSize = 1) THEN
						// Clear station output as occipied (to allow station to start oepration with only one station occupied)			
						afbStationCtrl[1].P_bVehicleReadyAtInput := FALSE;
					END_IF

					afbBufferControlPost[iBufferStation].M_AddVehicle(
														iVehicleID:= aStations[iBufferStation].stStationData2.nCurrentVehicleID, 
														iTicket:= aStations[iBufferStation].stStationData2.nTicket, 
														iTicketSize:= aStations[iBufferStation].stStationData2.nTicketSize, 
														iPriority:= aStations[iBufferStation].stStationData2.CurrentPriority, 
														iMoveCmdID:= iBufferMoveCmdID);
					aStations[iBufferStation].stStationData2.nTicket := 0;
					aStations[iBufferStation].stStationData2.nTicketSize := 0;
					aStations[iBufferStation].stStationData2.CurrentPriority := 0;
					aStations[iBufferStation].stStationData2.nCurrentVehicleID := 0;
					aStations[iBufferStation].stStationData2.nReservedVehicleID := 0;
					// signal movement finished
					afbStationCtrl[iBufferStation].bVehicleOutToPostMoved := TRUE;
					eBufferState := E_BufferState.FinishedOutToPost;
										
					F_LogLine('TC_BUF: Moving Out To Post-Buf CMD complete : %d', aStations[iBufferStation].stStationData2.nCurrentVehicleID);
				END_IF
				
			ELSIF (iRes = 3) THEN
				tonBuffersDelay.IN := FALSE;
				// Movement call failed... Retry
				
			END_IF
		END_IF

	E_BufferState.FinishedOutToPost:
		IF (NOT afbStationCtrl[iBufferStation].bMoveVehicleOutToPost) THEN
			afbStationCtrl[iBufferStation].bVehicleOutToPostMoved := FALSE;
			eBufferState := E_BufferState.Idle;
		END_IF

/////////////////////////////////////////////////////////////////////////////////////////////////////////////////////////////////////////////////////////
// Station input to post buffer
/////////////////////////////////////////////////////////////////////////////////////////////////////////////////////////////////////////////////////////		
	E_BufferState.MoveInToPost:
	// TODO!!! - Vehicle ID of vehicle in station OUT location?
		iRes := M_CallMoveVehicleToBuffer(	eInputType := E_MMVehicleInputType.eMMVehicleInputType_VehicleID, 
											sInput := UINT_TO_STRING(aStations[iBufferStation].stStationData1.nCurrentVehicleID), 
											sStationID := afbStationCtrl[iBufferStation].P_sStationID,
											eBufferType := E_MMStationBuffer.eMMStationBuffer_PostProcess, 
											nBufferIndex := TO_USINT(afbBufferControlPost[iBufferStation].P_iBufferSize), // Last location in buffer  
											eDirection := E_MMDirection.eMMDirection_Forward, 
											fVelocity := 0.5, 
											fAcceleration := 1,
											iCmdID => iBufferMoveCmdID 	);
		IF (iRes = 2) THEN
			// Movement call OK
			// Trig event-driven reading
			M_VehicleToReadAdd(aStations[iBufferStation].stStationData1.nCurrentVehicleID);
			F_LogLine('TC_BUF: Moving In To Post-Buf OK : %d', aStations[iBufferStation].stStationData1.nCurrentVehicleID);	
			eBufferState := E_BufferState.WaitInToPost;
		ELSIF (iRes = 3) THEN
			// Movement call failed
			// TODO!!!
			F_LogLine('TC_BUF: Error moving In To Post-Buf! : %d', aStations[iBufferStation].stStationData1.nCurrentVehicleID);
			eBufferState := E_BufferState.Idle;
		END_IF
	
	E_BufferState.WaitInToPost:
		tonBuffersDelay.IN := TRUE;
		tonBuffersDelay.PT := T#500MS;
		IF (tonBuffersDelay.Q) THEN
			iRes := M_CallMoveVehicleStatus(iCommandID := iBufferMoveCmdID,
											eMoveStatus => eBufferMoveState 	);
			IF (iRes = 2) THEN
				tonBuffersDelay.IN := FALSE;
				// Call OK
				IF (eBufferMoveState >= E_VehicleMoveState.ErrorLocation) THEN
					// Error with command
					// TODO!!!
					
				ELSIF (eBufferMoveState = E_VehicleMoveState.Moving OR eBufferMoveState = E_VehicleMoveState.Complete) THEN
					// Command completed!
					// Trig event-driven reading
					M_VehicleToReadAdd(aStations[iBufferStation].stStationData1.nCurrentVehicleID);				
				
					afbBufferControlPost[iBufferStation].M_AddVehicle(
														iVehicleID:= aStations[iBufferStation].stStationData1.nCurrentVehicleID, 
														iTicket:= aStations[iBufferStation].stStationData1.nTicket, 
														iTicketSize:= aStations[iBufferStation].stStationData1.nTicketSize, 
														iPriority:= aStations[iBufferStation].stStationData1.CurrentPriority, 
														iMoveCmdID:= iBufferMoveCmdID);
					aStations[iBufferStation].stStationData1.nTicket := 0;
					aStations[iBufferStation].stStationData1.nTicketSize := 0;
					aStations[iBufferStation].stStationData1.CurrentPriority := 0;
					aStations[iBufferStation].stStationData1.nCurrentVehicleID := 0;
					aStations[iBufferStation].stStationData1.nReservedVehicleID := 0;
					// signal movement finished
					afbStationCtrl[iBufferStation].bVehicleInToPostMoved := TRUE;
					eBufferState := E_BufferState.FinishedInToPost;
					
					F_LogLine('TC_BUF: Moving In To Post-Buf CMD complete : %d', aStations[iBufferStation].stStationData2.nCurrentVehicleID);
				END_IF
				
			ELSIF (iRes = 3) THEN
				tonBuffersDelay.IN := FALSE;
				// Movement call failed... Retry
				
			END_IF
		END_IF

	E_BufferState.FinishedInToPost:
		IF (NOT afbStationCtrl[iBufferStation].bMoveVehicleInToPost) THEN
			afbStationCtrl[iBufferStation].bVehicleInToPostMoved := FALSE;
			eBufferState := E_BufferState.Idle;
		END_IF
END_CASE

tonBuffersDelay(IN := ,
				PT := ,
				Q => ,
				ET => 	);
END_METHOD

/// Checks if any buffers are ready for the specified ticket and priority
/// Returns the station number which is ready to deliver vehicles from post buffer!
METHOD PROTECTED M_CTL_CheckStationsPostBuffer
VAR_INPUT
END_VAR
VAR_OUTPUT
	iTicket			: UINT;
	iStationID		: UINT;
	iBufferIndex	: UINT;
END_VAR
VAR
	i				: USINT;
	j				: USINT;
	iTicketSize		: UINT;
	iTicketCount	: UINT;
	iPostBufferSize	: UINT;
END_VAR
// Check if Vehicle can be used at stations 

// TODO!!! Handle multiple stations with priority!

iTicket := 0;
iTicketSize := 0;
iTicketCount := 0;

// NOTE: Only one station!!!
i := 2;

	// Check if station is active/present
	IF (afbStationCtrl[i].P_bPresent) THEN
		FOR j := MM_MAX_BUFFER_INDEX TO 1 BY -1 DO
			IF (aStations[i].astPostBuffer[j].bPresent) THEN
				// Check post buffer vehicles
				IF (aStations[i].astPostBuffer[j].nCurrentVehicleID > 0) THEN
					IF (iTicket = 0) THEN
						// First vehicle (closest to exit point in buffer)... Save ticket
						iTicket := aStations[i].astPostBuffer[j].nTicket;
						iTicketSize := aStations[i].astPostBuffer[j].nTicketSize;
						iTicketCount := iTicketCount+1;
					ELSE
						IF (aStations[i].astPostBuffer[j].nTicket = iTicket) THEN
							// One more vehicle with same ticket
							iTicketCount := iTicketCount+1;
							IF (iTicketCount >= iTicketSize) THEN
								// All with this ticket is ready in buffer. Release them
								iStationID := i;
								iBufferIndex := j;
								RETURN;
								
							ELSIF (j = 1) THEN
								// First index (closest to station) is reached
								// Check if another vehicle with same ticket is at the station
								IF (aStations[i].stStationData1.nTicket = iTicket) AND (afbStationCtrl[i].bCompletedInput OR afbStationCtrl[i].bCompletedOutput) THEN
									// Vehicle ready at station
									iStationID := i;
									iBufferIndex := j;
									RETURN;
									
								END_IF
							END_IF
						ELSE
							// New ticket, release the previous number of vehicles!
							iStationID := i;
							iBufferIndex := j;
							RETURN;
						END_IF
					END_IF
					
					// Check if vehicle Priority is the last on the ticket.
					IF (aStations[i].astPostBuffer[j].CurrentPriority >= aStations[i].astPostBuffer[j].nTicketSize) THEN
						iStationID := i;
						iBufferIndex := j;
						RETURN;
						
					END_IF
				ELSE
					// Empty buffer spot... Skip check
					iStationID := i;
					iBufferIndex := 0;
					RETURN;
				END_IF
			ELSIF (j = 1) THEN
				// No post buffer on the station... special Exit Point situation
				// (Use station location and pre buffer for check)
				// TODO!!!
			END_IF
		END_FOR
	END_IF
		

iTicket := 0;
iStationID := 0;
END_METHOD

/// Checks if any buffers are ready for the specified ticket and priority
METHOD PROTECTED M_CTL_CheckStationsPreBuffer
VAR_INPUT
	sStationID		: STRING(30);
	nVehicleID		: UINT;
	nTicket			: UINT;
	nPriority		: UINT;
END_VAR
VAR_OUTPUT
	nBufferIndex	: USINT;
END_VAR
VAR
	i				: USINT;
	iStat			: UINT;
	iBuf			: UINT;
END_VAR
//NO Pre buffer on stations for this cell

// Check if Vehicle can be used at stations 

// TODO!!! Handle multiple stations with priority!

//CASE eCellType OF
//	// Cell with own/separate track system
//	E_CellType.Type_Outline:
//		FOR i := 1 TO 5 BY 1 DO
//			// Check if station is active/present
//			IF (afbStationCtrl[i].P_bPresent) THEN
//				// Check if station has correct ID
//				IF (sStationID = afbStationCtrl[i].P_sStationID) THEN
//					// Check if station has free space in Pre-buffer
//					nBufferIndex := afbStationCtrl[i].M_AddVehicle(	nTicket := nTicket, 
//																	nVehicleID := nVehicleID, 
//																	nPriority := nPriority);
//					IF (nBufferIndex > 0) THEN
//						// Pre-Buffer space found, index saved in nBufferIndex
//						RETURN;	
//					END_IF
//				END_IF
//			ELSE
//				// No more stations present!
//				EXIT;
//			END_IF
//		END_FOR
	
//	// Cell located on main track system
//	E_CellType.Type_Inline:
//		FOR i := 1 TO 5 BY 1 DO
//			// Check if station is active/present
//			IF (afbStationCtrl[i].P_bPresent) THEN
//				// Check if station has correct ID
//				IF (sStationID = afbStationCtrl[i].P_sStationID) THEN
//					// Check if station has free space in Pre-buffer
//					nBufferIndex := afbStationCtrl[i].M_AddVehicle(	nTicket := nTicket, 
//																	nVehicleID := nVehicleID, 
//																	nPriority := nPriority);
//					IF (nBufferIndex > 0) THEN
//						// Pre-Buffer space found, index saved in nBufferIndex
//						RETURN;	
//					END_IF
//				END_IF
//			ELSE
//				// No more stations present!
//				EXIT;
//			END_IF
//		END_FOR
	
//	// Cell with only one track for both inlet and outlet
//	E_CellType.Type_InOut:
//		FOR i := 1 TO 5 BY 1 DO
//			// Check if station is active/present
//			IF (afbStationCtrl[i].P_bPresent) THEN
//				// Check if station has correct ID
//				IF (sStationID = afbStationCtrl[i].P_sStationID) THEN
//					// Check if station is occupied (only one ticket at a time to allow to move vehicles out of the cell after production
//					IF ( (aStations[i].stStationData1.nTicket = 0) OR (aStations[i].stStationData1.nTicket = nTicket) ) THEN  
//						// Check if station has free space in Pre-buffer
//						nBufferIndex := afbStationCtrl[i].M_AddVehicle(	nTicket := nTicket, 
//																		nVehicleID := nVehicleID, 
//																		nPriority := nPriority);
//						IF (nBufferIndex > 0) THEN
//							// Pre-Buffer space found, index saved in nBufferIndex
//							RETURN;	
//						END_IF
//					END_IF
//				END_IF
//			ELSE
//				// No more stations present!
//				EXIT;
//			END_IF
//		END_FOR

//END_CASE
END_METHOD

METHOD PROTECTED M_CTL_CheckTicket : BOOL
VAR_INPUT
	nTicket			: UINT;
END_VAR
VAR
	i				: UINT;
	bFound			: BOOL;
END_VAR

bFound := FALSE;

// Check if the specified ticket is expected at the specified station
FOR i := 1 TO MM_MAX_RESERVATIONLIST_ELEMENTS BY 1 DO
	IF (aReadCellData.stCell.astReservations[i].nTicket = nTicket) THEN
		// Set found status and exit FOR loop
		bFound := TRUE;
		EXIT;
	END_IF
END_FOR

// return status
M_CTL_CheckTicket := bFound;
END_METHOD

METHOD PROTECTED M_CTL_DecisionPoint : BOOL
VAR_INPUT
END_VAR
VAR
	i					: INT;
	iRes				: INT;
	sTempString			: STRING(200);
END_VAR
VAR 
END_VAR

